      CALL FC   563 (
           ActReq                   := M    101.0,
           PLCNo                    := DB1575.DBW   14,
           SourceUnitNo             := 91,
           IsTUnit                  := FALSE,
           DstComDRec               := DB1575.CIP,
           RET_VAL                  := #wRetVal);


// ... CIP Distribution ------------- /

      L     DB1571.DBD   46;
      L     DB1945.DBD   10;
      ==D   ;
      JCN   CIP1;
      CALL FC   563 (
           ActReq                   := M    101.0,
           PLCNo                    := 3,
           SourceUnitNo             := 91,
           IsTUnit                  := FALSE,
           DstComDRec               := DB1575.CIP,
           RET_VAL                  := #wRetVal);

      CALL FC   563 (
           ActReq                   := M    101.0,
           PLCNo                    := 3,
           SourceUnitNo             := 94,
           IsTUnit                  := FALSE,
           DstComDRec               := DB1575.CIPDist,
           RET_VAL                  := #wRetVal);

      CALL SFC   20 (
           SRCBLK                   := DB1575.ToCIP,
           RET_VAL                  := #iRetVal,
           DSTBLK                   := DB502.ToCIP1);

CIP1: NOP   0;

      L     DB1571.DBD   46;
      L     DB1955.DBD   10;
      ==D   ;
      JCN   CIP2;
      CALL FC   563 (
           ActReq                   := M    101.0,
           PLCNo                    := 3,
           SourceUnitNo             := 92,
           IsTUnit                  := FALSE,
           DstComDRec               := DB1575.CIP,
           RET_VAL                  := #wRetVal);

      CALL FC   563 (
           ActReq                   := M    101.0,
           PLCNo                    := 3,
           SourceUnitNo             := 95,
           IsTUnit                  := FALSE,
           DstComDRec               := DB1575.CIPDist,
           RET_VAL                  := #wRetVal);

      CALL SFC   20 (
           SRCBLK                   := DB1575.ToCIP,
           RET_VAL                  := #iRetVal,
           DSTBLK                   := DB502.ToCIP2);
CIP2: NOP   0;

      L     DB1571.DBD   46;
      L     DB1965.DBD   10;
      ==D   ;
      JCN   CIP3;
      CALL FC   563 (
           ActReq                   := M    101.0,
           PLCNo                    := 3,
           SourceUnitNo             := 93,
           IsTUnit                  := FALSE,
           DstComDRec               := DB1575.CIP,
           RET_VAL                  := #wRetVal);

      CALL FC   563 (
           ActReq                   := M    101.0,
           PLCNo                    := 3,
           SourceUnitNo             := 96,
           IsTUnit                  := FALSE,
           DstComDRec               := DB1575.CIPDist,
           RET_VAL                  := #wRetVal);

      CALL SFC   20 (
           SRCBLK                   := DB1575.ToCIP,
           RET_VAL                  := #iRetVal,
           DSTBLK                   := DB502.ToCIP3);

CIP3: NOP   0;

//----------------------------------------
// Communication Water Tank
//----------------------------------------
// Current Tank ----------------------------
      CALL FC   950 (
           EquipmentNo              := DB1571.DBD  270,
           PLCNo                    := #iPLC,
           UnitNo                   := #iUnit);
      L     #iUnit;
      L     0;
      >I    ;
      JCN   T0xx;

      CALL FC   563 (
           ActReq                   := M    101.0,
           PLCNo                    := #iPLC,
           SourceUnitNo             := #iUnit,
           IsTUnit                  := FALSE,
           DstComDRec               := DB1575.SRC,
           RET_VAL                  := #wRetVal);
      JU    T0xy;
T0xx: NOP   0;
      T     #iTmp;
      CALL SFC   21 (
           BVAL                     := #iTmp,
           RET_VAL                  := #iRetVal,
           BLK                      := DB1575.SRC);
T0xy: NOP   0;

// Priority 1 -----------------------------
      CALL FC   950 (
           EquipmentNo              := DB1571.DBD  286,
           PLCNo                    := #iPLC,
           UnitNo                   := #iUnit);
      L     #iUnit;
      L     0;
      >I    ;
      JCN   T1xx;

      CALL FC   563 (
           ActReq                   := M    101.0,
           PLCNo                    := #iPLC,
           SourceUnitNo             := #iUnit,
           IsTUnit                  := FALSE,
           DstComDRec               := DB1575.SRC1,
           RET_VAL                  := #wRetVal);
      JU    T1xy;
T1xx: NOP   0;
      T     #iTmp;
      CALL SFC   21 (
           BVAL                     := #iTmp,
           RET_VAL                  := #iRetVal,
           BLK                      := DB1575.SRC1);
T1xy: NOP   0;

// Priority 2 ----------------------------
      CALL FC   950 (
           EquipmentNo              := DB1571.DBD  302,
           PLCNo                    := #iPLC,
           UnitNo                   := #iUnit);
      L     #iUnit;
      L     0;
      >I    ;
      JCN   T2xx;

      CALL FC   563 (
           ActReq                   := M    101.0,
           PLCNo                    := #iPLC,
           SourceUnitNo             := #iUnit,
           IsTUnit                  := FALSE,
           DstComDRec               := DB1575.SRC2,
           RET_VAL                  := #wRetVal);
      JU    T2xy;
T2xx: NOP   0;
      T     #iTmp;
      CALL SFC   21 (
           BVAL                     := #iTmp,
           RET_VAL                  := #iRetVal,
           BLK                      := DB1575.SRC2);
T2xy: NOP   0;

// Pririty 3 ----------------------------
      CALL FC   950 (
           EquipmentNo              := DB1571.DBD  318,
           PLCNo                    := #iPLC,
           UnitNo                   := #iUnit);
      L     #iUnit;
      L     0;
      >I    ;
      JCN   T3xx;

      CALL FC   563 (
           ActReq                   := M    101.0,
           PLCNo                    := #iPLC,
           SourceUnitNo             := #iUnit,
           IsTUnit                  := FALSE,
           DstComDRec               := DB1575.SRC3,
           RET_VAL                  := #wRetVal);
      JU    T3xy;
T3xx: NOP   0;
      T     #iTmp;
      CALL SFC   21 (
           BVAL                     := #iTmp,
           RET_VAL                  := #iRetVal,
           BLK                      := DB1575.SRC3);
T3xy: NOP   0;

//----------------------------------------
// Communication Brewhouse
//----------------------------------------
///   L     #U.Seq.Prop.Index0          // Destination
///   ITD
///   DTR
///   T     #rTmp

///  CALL  "Eq2PU"
//       EquipmentNo:=#rTmp
//       PLCNo      :=#iPLC
//       UnitNo     :=#iUnit

///  CALL  "UIT3"
//       ActReq      :="Clk1E"
//       PLCNo       :=#iPLC
//       SourceUnitNo:=#iUnit
//       IsTUnit     :=FALSE
//       DstComDRec  :="C04ComD".DST
//       RET_VAL     :=#wRetVal



NETWORK
TITLE =remote start

      SET   ;
// !!! insert correct condition of unit start !!!
      A     DB1571.DBX   15.0;
      A     DB1571.DBX   17.4;
      CLR   ;
      JCN   Strt;
      L     DB1575.DBD   10;
//L        L#-1;                            // Prid negative to start on its own
      T     #Prid;

      CALL FC    48 (
           UnitNo                   := #UnitNo,
           PrId                     := #Prid,
           Run                      := DB1571.DBX   17.4,
           PrIdTransfer             := TRUE,
           Start                    := TRUE,
           RetVal                   := #wRetVal);
Strt: NOP   0;
NETWORK
TITLE =external releases

      SET   ;
      =     DB2570.DBX  106.7;
      =     DB2570.DBX  426.7;
      =     DB2570.DBX  506.7;

NETWORK
TITLE =write own unit data

      SET   ;

//-- CIP Communication ---------------------------------------
      AN    DB1571.DBX   15.0;
//      AN "U057SeqD".Seq.PO.B30 // CIP Active (Slave)
      A     #ComCIP;
      JCN   NCIP;
//Conductivity CIP Return
      L     DB1575.DBD  150;
      T     DB1571.DBD  626;

//Temperature CIP Return
      L     DB1575.DBD  146;
      T     DB1571.DBD  594;

//CIP Prerun Pump SP

      CALL FC    45 (
           SFM                      := DB1571.DBD  686,
           Indexes                  := #SFM36);


      L     0.000000e+000;
      A     #SFM36.I01;
      =     DB1575.DBX  171.7;
      JCN   pfc;
      L     DB1571.DBD  654;
pfc:  NOP   0;
      A     #SFM36.I02;
      =     DB1575.DBX  172.0;
      JCN   ppc;
      L     DB1571.DBD  670;
ppc:  NOP   0;
      A     #SFM36.I03;
      =     DB1575.DBX  171.6;
      JCN   pxc;
      L     DB1571.DBD  574;
pxc:  NOP   0;
      T     DB1575.DBD  182;

//CIP Return
      L     DB1571.DBD  558;
      T     DB1575.DBD  186;
      L     DB1575.DBD  138;
      T     DB1571.DBD  562;

//CIP Prerun
      L     DB1571.DBD  542;
      T     DB1575.DBD  190;
      L     DB1575.DBD  142;
      T     DB1571.DBD  546;

// Write Own Data to CIP
      L     DB1575.DBD   10;
      T     DB1575.DBD  154;

      L     DB1575.DBW   14;
      T     DB1575.DBW  158;

      L     DB1575.DBW   16;
      T     DB1575.DBW  160;

      L     DB1575.DBW   18;
      T     DB1575.DBW  162;

      L     DB1575.DBW   20;
      T     DB1575.DBW  164;

      L     DB1575.DBW   22;
      T     DB1575.DBW  166;

      A     DB1575.DBX   24.0;
      =     DB1575.DBX  168.0;

      A     DB1575.DBX   24.1;
      =     DB1575.DBX  168.1;

      A     DB1575.DBX   24.2;
      =     DB1575.DBX  168.2;

      A     DB1575.DBX   24.3;
      =     DB1575.DBX  168.3;

      A     DB1575.DBX   24.4;
      =     DB1575.DBX  168.4;

      A     DB1575.DBX   24.5;
      =     DB1575.DBX  168.5;

      A     DB1575.DBX   24.6;
      =     DB1575.DBX  168.6;

      A     DB1575.DBX   24.7;
      =     DB1575.DBX  168.7;

// Copy Data to CIP
      CALL SFC   20 (
           SRCBLK                   := DB1575.ToCIP,
           RET_VAL                  := #iRetVal,
           DSTBLK                   := DB1575.ToCIP);

NCIP: NOP   0;

//Empty Signal
//A     "U057SpID".SpI.Sig //!!!! Insert correct Empty Signal !!!
      CLR   ;
      =     DB1575.DBX   26.5;

//Full Signal
//A     "U057SpID".SpI.Sig //!!!! Insert correct Full Signal !!!
      CLR   ;
      =     DB1575.DBX   26.2;

//CIP Program Selected
      A     #CIP;
      =     DB1575.DBX   27.1;

// Emergency Stop
      A     #EStopOK; //If needed add or replace with own SpI
      =     DB1575.DBX   27.0; //Emergency Stop OK

      L     DB1571.DBD  782; // Material
      T     DB1575.DBD   30;

      L     DB1571.DBD  270; // Current Water Tank Selection
      T     DB1575.DBD   34;

      L     DB1571.DBD  286; // Priority 1
      T     DB1575.DBD   38;

      L     DB1571.DBD  302; // Priority 2
      T     DB1575.DBD   42;

      L     DB1571.DBD  318; // Priority 3
      T     DB1575.DBD   46;

NETWORK
TITLE = read from other unit data



END_FUNCTION_BLOCK

FUNCTION_BLOCK FB 1579
TITLE =U057: Water Transfer Brewhouse
AUTHOR : Woermann
FAMILY : BOTEC_F1
NAME : Sim
VERSION : 0.1


VAR_TEMP
  CIP : BOOL ;	//CIP active
  xTmp : BOOL ;	//Temporary BOOL (free for general use)
  iTmp : INT ;	//Temporary INT (free for general use)
  rTmp : REAL ;	//Temporary REAL (free for general use)
  UnitNo : INT ;	//Unit Number
END_VAR
BEGIN
NETWORK
TITLE =General

      SET   ;
// get unit number ----------------------------------------------------------
      L     DB1570.DBW    0;
      T     #UnitNo;

// CIP ----------------------------------------------------------------------
      L     DB1571.DBD   54;
      L     0;
      <D    ;
      =     #CIP;

NETWORK
TITLE =Actuator

      A     DB1571.DBX   17.3;
      =     DB2570.DBX  105.3;
      =     DB2570.DBX  185.3;
      =     DB2570.DBX  265.3;
      =     DB2570.DBX  345.3;
      =     DB2570.DBX  505.3;


NETWORK
TITLE =Special Input

      A     DB1571.DBX   17.3;
      =     DB2571.DBX  141.3;
      =     DB2571.DBX  201.3;
      =     DB2571.DBX  261.3;
      =     DB2571.DBX  321.3;
      =     DB2571.DBX  381.3;

NETWORK
TITLE =Counter

      A     DB1571.DBX   17.3;
      A     M    101.0;


      CLR   ;
NETWORK
TITLE =Analog Input

      A     DB1571.DBX   17.3;

NETWORK
TITLE =Universal Value

      A     DB1571.DBX   17.3;
//      =     "U057UnVD".unv001.Sim;
//      =     "U057UnVD".unv002.Sim;
//      =     "U057UnVD".unv003.Sim;
//      =     "U057UnVD".unv004.Sim;

NETWORK
TITLE =PID

      A     DB1571.DBX   17.3;

NETWORK
TITLE =Message

      A     DB1571.DBX   17.3;
//      =     "U057MsgD".msg001.Sim;
//      =     "U057MsgD".msg002.Sim;
//      =     "U057MsgD".msg003.Sim;

NETWORK
TITLE =VLT

      A     DB1571.DBX   17.3;

END_FUNCTION_BLOCK

FUNCTION_BLOCK FB 1585
TITLE =U058: Water Transfer Syrup
FAMILY : BOTEC_F1
NAME : Comm
VERSION : 0.1


VAR_TEMP
  iRetVal : INT ;	//return value as integer
  wRetVal : WORD ;	//return value as word
  Run : BOOL ;	//Unit in "RUN" mode
  EStopOK : BOOL ;	//Emergency Stop OK
  CIP : BOOL ;	//CIP Program Selected
  ComCIP : BOOL ;	//Communication with CIP Active
  xTmp : BOOL ;	//Temporary BOOL (free for general use)
  iTmp : INT ;	//Temporary INT (free for general use)
  rTmp : REAL ;	//Temporary REAL (free for general use)
  dTmp : DINT ;	//Temporary DINT (free for general use)
  UnitNo : INT ;	//Unit Number
  EquipmentID : INT ;	//Equipment ID
  Prid : DINT ;	//Process ID
  SFM36 : STRUCT 	// CIP Pump Mode
   I00 : BOOL ;	// Off
   I01 : BOOL ;	// Flow
   I02 : BOOL ;	// Pressure
   I03 : BOOL ;	// Fix Speed
   I04 : BOOL ;
   I05 : BOOL ;
   I06 : BOOL ;
   I07 : BOOL ;
   I08 : BOOL ;
   I09 : BOOL ;
   I10 : BOOL ;
   I11 : BOOL ;
   I12 : BOOL ;
   I13 : BOOL ;
   I14 : BOOL ;
   I15 : BOOL ;
   I16 : BOOL ;
   I17 : BOOL ;
   I18 : BOOL ;
   I19 : BOOL ;
   I20 : BOOL ;
   I21 : BOOL ;
   I22 : BOOL ;
   I23 : BOOL ;
   I24 : BOOL ;
   I25 : BOOL ;
   I26 : BOOL ;
   I27 : BOOL ;
   I28 : BOOL ;
   I29 : BOOL ;
   I30 : BOOL ;
   I31 : BOOL ;
  END_STRUCT ;
  iPLC : INT ;
  iUnit : INT ;
END_VAR
BEGIN
NETWORK
TITLE =general

      SET   ;

// unit & equipment number ---------------------------------------------------
      L     DB1580.DBW    0;
      T     #UnitNo;

      L     DB1585.DBW   14;
      L     1000;
      *I    ;
      L     #UnitNo;
      +I    ;
      T     #EquipmentID;

// CIP ----------------------------------------------------------------------
      L     DB1585.DBW   18;
      L     0;
      <I    ;
      =     #CIP;

// Communicating Units-------------------------------------------------------
      L     DB1585.DBD   10;
      L     DB1585.DBD  106;
      ==D   ;
      =     #ComCIP;

// emergency OK -------------------------------------------------------------
      A     DB1585.DBX   75.0; //General Emergency Stop OK
      =     #EStopOK;

NETWORK
TITLE =read other unit's data

      SET   ;

// ... General Unit ----------/

      CALL FC   563 (
           ActReq                   := M    101.0,
           PLCNo                    := DB1585.DBW   14,
           SourceUnitNo             := 99,
           IsTUnit                  := FALSE,
           DstComDRec               := DB1585.GEN,
           RET_VAL                  := #wRetVal);


// ... CIP Unit ------------- /

      CALL FC   563 (
           ActReq                   := M    101.0,
           PLCNo                    := DB1585.DBW   14,
           SourceUnitNo             := 92,
           IsTUnit                  := FALSE,
           DstComDRec               := DB1585.CIP,
           RET_VAL                  := #wRetVal);


// ... CIP Distribution ------------- /
      L     DB1581.DBD   46;
      L     DB1955.DBD   10;
      ==D   ;
      JCN   CIP2;

      CALL FC   563 (
           ActReq                   := M    101.0,
           PLCNo                    := 3,
           SourceUnitNo             := 95,
           IsTUnit                  := FALSE,
           DstComDRec               := DB1585.CIPDist,
           RET_VAL                  := #wRetVal);

      CALL SFC   20 (
           SRCBLK                   := DB1585.ToCIP,
           RET_VAL                  := #iRetVal,
           DSTBLK                   := DB502.ToCIP2);
CIP2: NOP   0;

//----------------------------------------
// Communication Water Tank
//----------------------------------------
// Current Tank ----------------------------
      CALL FC   950 (
           EquipmentNo              := DB1581.DBD  270,
           PLCNo                    := #iPLC,
           UnitNo                   := #iUnit);
      L     #iUnit;
      L     0;
      >I    ;
      JCN   T0xx;
      CALL FC   563 (
           ActReq                   := M    101.0,
           PLCNo                    := #iPLC,
           SourceUnitNo             := #iUnit,
           IsTUnit                  := FALSE,
           DstComDRec               := DB1585.SRC,
           RET_VAL                  := #wRetVal);
      JU    T0xy;
T0xx: NOP   0;
      T     #iTmp;
      CALL SFC   21 (
           BVAL                     := #iTmp,
           RET_VAL                  := #iRetVal,
           BLK                      := DB1585.SRC);
T0xy: NOP   0;

// Priority 1 -----------------------------
      CALL FC   950 (
           EquipmentNo              := DB1581.DBD  286,
           PLCNo                    := #iPLC,
           UnitNo                   := #iUnit);
      L     #iUnit;
      L     0;
      >I    ;
      JCN   T1xx;

      CALL FC   563 (
           ActReq                   := M    101.0,
           PLCNo                    := #iPLC,
           SourceUnitNo             := #iUnit,
           IsTUnit                  := FALSE,
           DstComDRec               := DB1585.SRC1,
           RET_VAL                  := #wRetVal);
      JU    T1xy;
T1xx: NOP   0;
      T     #iTmp;
      CALL SFC   21 (
           BVAL                     := #iTmp,
           RET_VAL                  := #iRetVal,
           BLK                      := DB1585.SRC1);
T1xy: NOP   0;

// Priority 2 ----------------------------
      CALL FC   950 (
           EquipmentNo              := DB1581.DBD  302,
           PLCNo                    := #iPLC,
           UnitNo                   := #iUnit);
      L     #iUnit;
      L     0;
      >I    ;
      JCN   T2xx;

      CALL FC   563 (
           ActReq                   := M    101.0,
           PLCNo                    := #iPLC,
           SourceUnitNo             := #iUnit,
           IsTUnit                  := FALSE,
           DstComDRec               := DB1585.SRC2,
           RET_VAL                  := #wRetVal);
      JU    T2xy;
T2xx: NOP   0;
      T     #iTmp;
      CALL SFC   21 (
           BVAL                     := #iTmp,
           RET_VAL                  := #iRetVal,
           BLK                      := DB1585.SRC2);
T2xy: NOP   0;

// Pririty 3 ----------------------------
      CALL FC   950 (
           EquipmentNo              := DB1581.DBD  318,
           PLCNo                    := #iPLC,
           UnitNo                   := #iUnit);
      L     #iUnit;
      L     0;
      >I    ;
      JCN   T3xx;

      CALL FC   563 (
           ActReq                   := M    101.0,
           PLCNo                    := #iPLC,
           SourceUnitNo             := #iUnit,
           IsTUnit                  := FALSE,
           DstComDRec               := DB1585.SRC3,
           RET_VAL                  := #wRetVal);
      JU    T3xy;
T3xx: NOP   0;
      T     #iTmp;
      CALL SFC   21 (
           BVAL                     := #iTmp,
           RET_VAL                  := #iRetVal,
           BLK                      := DB1585.SRC3);
T3xy: NOP   0;


// Sirupraum
      CALL FC   563 (
           ActReq                   := M    101.0,
           PLCNo                    := 1,
           SourceUnitNo             := 8,
           IsTUnit                  := FALSE,
           DstComDRec               := DB1585.DST,
           RET_VAL                  := #wRetVal);

NETWORK
TITLE =remote start

      SET   ;
// !!! insert correct condition of unit start !!!
      A     DB1581.DBX   15.0;
      A     DB1581.DBX   17.4;
      CLR   ;
      JCN   Strt;
      L     DB1585.DBD   10;
//L        L#-1;                            // Prid negative to start on its own
      T     #Prid;

      CALL FC    48 (
           UnitNo                   := #UnitNo,
           PrId                     := #Prid,
           Run                      := DB1581.DBX   17.4,
           PrIdTransfer             := TRUE,
           Start                    := TRUE,
           RetVal                   := #wRetVal);
Strt: NOP   0;
NETWORK
TITLE =external releases

      SET   ;
      =     DB2580.DBX  106.7;
      =     DB2580.DBX  186.7;
      =     DB2580.DBX  266.7;
NETWORK
TITLE =write own unit data

      SET   ;

//-- CIP Communication ---------------------------------------
      AN    DB1581.DBX   15.0;
//      AN "U058SeqD".Seq.PO.B30 // CIP Active (Slave)
      A     #ComCIP;
      JCN   NCIP;
//Conductivity CIP Return
      L     DB1585.DBD  150;
      T     DB1581.DBD  626;

//Temperature CIP Return
      L     DB1585.DBD  146;
      T     DB1581.DBD  594;

//CIP Prerun Pump SP

      CALL FC    45 (
           SFM                      := DB1581.DBD  686,
           Indexes                  := #SFM36);


      L     0.000000e+000;
      A     #SFM36.I01;
      =     DB1585.DBX  171.7;
      JCN   pfc;
      L     DB1581.DBD  654;
pfc:  NOP   0;
      A     #SFM36.I02;
      =     DB1585.DBX  172.0;
      JCN   ppc;
      L     DB1581.DBD  670;
ppc:  NOP   0;
      A     #SFM36.I03;
      =     DB1585.DBX  171.6;
      JCN   pxc;
      L     DB1581.DBD  574;
pxc:  NOP   0;
      T     DB1585.DBD  182;

//CIP Return
      L     DB1581.DBD  558;
      T     DB1585.DBD  186;
      L     DB1585.DBD  138;
      T     DB1581.DBD  562;

//CIP Prerun
      L     DB1581.DBD  542;
      T     DB1585.DBD  190;
      L     DB1585.DBD  142;
      T     DB1581.DBD  546;

// Write Own Data to CIP
      L     DB1585.DBD   10;
      T     DB1585.DBD  154;

      L     DB1585.DBW   14;
      T     DB1585.DBW  158;

      L     DB1585.DBW   16;
      T     DB1585.DBW  160;

      L     DB1585.DBW   18;
      T     DB1585.DBW  162;

      L     DB1585.DBW   20;
      T     DB1585.DBW  164;

      L     DB1585.DBW   22;
      T     DB1585.DBW  166;

      A     DB1585.DBX   24.0;
      =     DB1585.DBX  168.0;

      A     DB1585.DBX   24.1;
      =     DB1585.DBX  168.1;

      A     DB1585.DBX   24.2;
      =     DB1585.DBX  168.2;

      A     DB1585.DBX   24.3;
      =     DB1585.DBX  168.3;

      A     DB1585.DBX   24.4;
      =     DB1585.DBX  168.4;

      A     DB1585.DBX   24.5;
      =     DB1585.DBX  168.5;

      A     DB1585.DBX   24.6;
      =     DB1585.DBX  168.6;

      A     DB1585.DBX   24.7;
      =     DB1585.DBX  168.7;

// Copy Data to CIP
      CALL SFC   20 (
           SRCBLK                   := DB1585.ToCIP,
           RET_VAL                  := #iRetVal,
           DSTBLK                   := DB502.ToCIP2);

NCIP: NOP   0;

//Empty Signal
//A     "U058SpID".SpI.Sig //!!!! Insert correct Empty Signal !!!
      CLR   ;
      =     DB1585.DBX   26.5;

//Full Signal
//A     "U058SpID".SpI.Sig //!!!! Insert correct Full Signal !!!
      CLR   ;
      =     DB1585.DBX   26.2;

//CIP Program Selected
      A     #CIP;
      =     DB1585.DBX   27.1;

// Emergency Stop
      A     #EStopOK; //If needed add or replace with own SpI
      =     DB1585.DBX   27.0; //Emergency Stop OK

// Weitere Signale
      L     DB1581.DBD  782; // Material
      T     DB1585.DBD   30;

      L     DB1581.DBD  270; // Current Water Tank Selection
      T     DB1585.DBD   34;

      L     DB1581.DBD  286; // Priority 1
      T     DB1585.DBD   38;

      L     DB1581.DBD  302; // Priority 2
      T     DB1585.DBD   42;

      L     DB1581.DBD  318; // Priority 3
      T     DB1585.DBD   46;



      A     DB1585.DBX  458.1;
      ON    DB5030.DBX  182.5;
      ON    DB5050.DBX  182.5;
      ON    DB5070.DBX  182.5;
      ON    DB5090.DBX  182.5;
      ON    DB5120.DBX  182.5;
      ON    DB5140.DBX  182.5;
      =     DB1585.DBX   26.3;


NETWORK
TITLE = read from other unit data



END_FUNCTION_BLOCK

FUNCTION_BLOCK FB 1589
TITLE =U058: Water Transfer Syrup
AUTHOR : Woermann
FAMILY : BOTEC_F1
NAME : Sim
VERSION : 0.1


VAR_TEMP
  CIP : BOOL ;	//CIP active
  xTmp : BOOL ;	//Temporary BOOL (free for general use)
  iTmp : INT ;	//Temporary INT (free for general use)
  rTmp : REAL ;	//Temporary REAL (free for general use)
  UnitNo : INT ;	//Unit Number
END_VAR
BEGIN
NETWORK
TITLE =General

      SET   ;
// get unit number ----------------------------------------------------------
      L     DB1580.DBW    0;
      T     #UnitNo;

// CIP ----------------------------------------------------------------------
      L     DB1581.DBD   54;
      L     0;
      <D    ;
      =     #CIP;

NETWORK
TITLE =Actuator

      A     DB1581.DBX   17.3;
      =     DB2580.DBX  105.3;
      =     DB2580.DBX  185.3;
      =     DB2580.DBX  265.3;
      =     DB2580.DBX  505.3;

NETWORK
TITLE =Special Input

      A     DB1581.DBX   17.3;
      =     DB2581.DBX  141.3;
      =     DB2581.DBX  201.3;


NETWORK
TITLE =Counter

      A     DB1581.DBX   17.3;
      A     M    101.0;


      CLR   ;
NETWORK
TITLE =Analog Input

      A     DB1581.DBX   17.3;
      =     DB2583.DBX  141.3;

NETWORK
TITLE =Universal Value

      A     DB1581.DBX   17.3;
//      =     "U058UnVD".unv001.Sim;
//      =     "U058UnVD".unv002.Sim;
//      =     "U058UnVD".unv003.Sim;
//      =     "U058UnVD".unv004.Sim;

NETWORK
TITLE =PID

      A     DB1581.DBX   17.3;
//      =     "U058PIDD".SR_P1_PID.Ign;

NETWORK
TITLE =Message

      A     DB1581.DBX   17.3;
//      =     "U058MsgD".msg001.Sim;
//      =     "U058MsgD".msg002.Sim;
//      =     "U058MsgD".msg003.Sim;

NETWORK
TITLE =VLT

      A     DB1581.DBX   17.3;

END_FUNCTION_BLOCK

FUNCTION_BLOCK FB 1595
TITLE =U059: Molchwasser
FAMILY : BOTEC_F1
NAME : U059Comm
VERSION : 0.1


VAR_TEMP
  iRetVal : INT ;	//return value as integer
  wRetVal : WORD ;	//return value as word
  Run : BOOL ;	//Unit in "RUN" mode
  EStopOK : BOOL ;	//Emergency Stop OK
  CIP : BOOL ;	//CIP Program Selected
  ComCIP : BOOL ;	//Communication with CIP Active
  xTmp : BOOL ;	//Temporary BOOL (free for general use)
  iTmp : INT ;	//Temporary INT (free for general use)
  rTmp : REAL ;	//Temporary REAL (free for general use)
  dTmp : DINT ;	//Temporary DINT (free for general use)
  UnitNo : INT ;	//Unit Number
  EquipmentID : INT ;	//Equipment ID
  Prid : DINT ;	//Process ID
  SFM36 : STRUCT 	// CIP Pump Mode
   I00 : BOOL ;	// Off
   I01 : BOOL ;	// Flow
   I02 : BOOL ;	// Pressure
   I03 : BOOL ;	// Fix Speed
   I04 : BOOL ;
   I05 : BOOL ;
   I06 : BOOL ;
   I07 : BOOL ;
   I08 : BOOL ;
   I09 : BOOL ;
   I10 : BOOL ;
   I11 : BOOL ;
   I12 : BOOL ;
   I13 : BOOL ;
   I14 : BOOL ;
   I15 : BOOL ;
   I16 : BOOL ;
   I17 : BOOL ;
   I18 : BOOL ;
   I19 : BOOL ;
   I20 : BOOL ;
   I21 : BOOL ;
   I22 : BOOL ;
   I23 : BOOL ;
   I24 : BOOL ;
   I25 : BOOL ;
   I26 : BOOL ;
   I27 : BOOL ;
   I28 : BOOL ;
   I29 : BOOL ;
   I30 : BOOL ;
   I31 : BOOL ;
  END_STRUCT ;
END_VAR
BEGIN
NETWORK
TITLE =general

      SET   ;

// unit & equipment number ---------------------------------------------------
      L     DB1590.DBW    0;
      T     #UnitNo;

      L     DB1595.DBW   14;
      L     1000;
      *I    ;
      L     #UnitNo;
      +I    ;
      T     #EquipmentID;

// CIP ----------------------------------------------------------------------
      L     DB1595.DBW   18;
      L     0;
      <I    ;
      =     #CIP;

// Communicating Units-------------------------------------------------------
      L     DB1595.DBD   10;
      L     DB1595.DBD  106;
      ==D   ;
      =     #ComCIP;

// emergency OK -------------------------------------------------------------
      A     DB1595.DBX   75.0; //General Emergency Stop OK
      =     #EStopOK;

NETWORK
TITLE =read other unit's data

      SET   ;

// ... General Unit ----------/

      CALL FC   563 (
           ActReq                   := M    101.0,
           PLCNo                    := 3,
           SourceUnitNo             := 99,
           IsTUnit                  := FALSE,
           DstComDRec               := DB1595.GEN,
           RET_VAL                  := #wRetVal);


NETWORK
TITLE =remote start
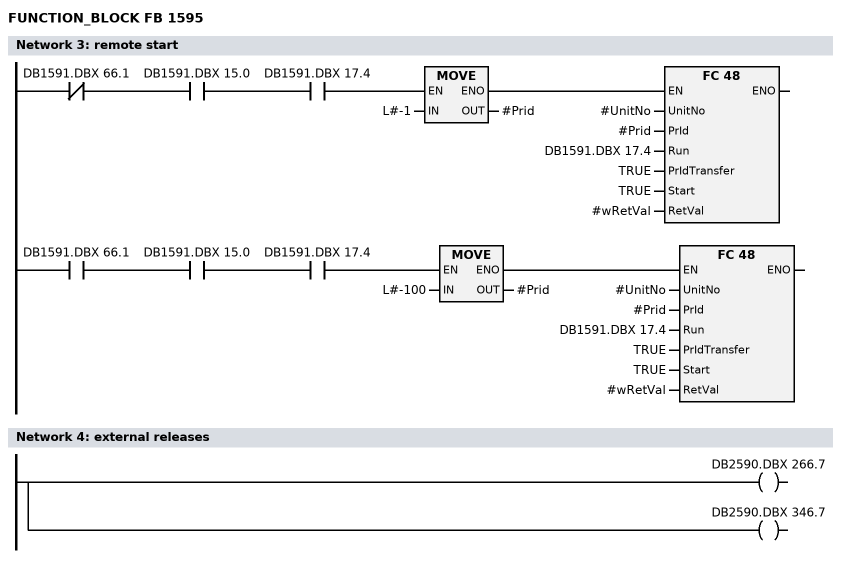

      SET   ;
      AN    DB1591.DBX   66.1;
      A     DB1591.DBX   15.0;
      A     DB1591.DBX   17.4;
      JCN   Strt;
      L     L#-1; // Prid negative to start on its own
      T     #Prid;

      CALL FC    48 (
           UnitNo                   := #UnitNo,
           PrId                     := #Prid,
           Run                      := DB1591.DBX   17.4,
           PrIdTransfer             := TRUE,
           Start                    := TRUE,
           RetVal                   := #wRetVal);
Strt: NOP   0;

      A     DB1591.DBX   66.1;
      A     DB1591.DBX   15.0;
      A     DB1591.DBX   17.4;
      JCN   Str2;
      L     L#-100; // Prid negative to start on its own
      T     #Prid;

      CALL FC    48 (
           UnitNo                   := #UnitNo,
           PrId                     := #Prid,
           Run                      := DB1591.DBX   17.4,
           PrIdTransfer             := TRUE,
           Start                    := TRUE,
           RetVal                   := #wRetVal);
Str2: NOP   0;

NETWORK
TITLE =external releases

      SET   ;
      =     DB2590.DBX  266.7;
      =     DB2590.DBX  346.7;
NETWORK
TITLE =write own unit data

      SET   ;

//-- CIP Communication ---------------------------------------
      AN    DB1591.DBX   15.0;
//      AN "U059SeqD".Seq.PO.B30 // CIP Active (Slave)
      A     #ComCIP;
      JCN   NCIP;
//Conductivity CIP Return
      L     DB1595.DBD  150;
      T     DB1591.DBD  626;

//Temperature CIP Return
      L     DB1595.DBD  146;
      T     DB1591.DBD  594;

//CIP Prerun Pump SP

      CALL FC    45 (
           SFM                      := DB1591.DBD  686,
           Indexes                  := #SFM36);


      L     0.000000e+000;
      A     #SFM36.I01;
      =     DB1595.DBX  171.7;
      JCN   pfc;
      L     DB1591.DBD  654;
pfc:  NOP   0;
      A     #SFM36.I02;
      =     DB1595.DBX  172.0;
      JCN   ppc;
      L     DB1591.DBD  670;
ppc:  NOP   0;
      A     #SFM36.I03;
      =     DB1595.DBX  171.6;
      JCN   pxc;
      L     DB1591.DBD  574;
pxc:  NOP   0;
      T     DB1595.DBD  182;

//CIP Return
      L     DB1591.DBD  558;
      T     DB1595.DBD  186;
      L     DB1595.DBD  138;
      T     DB1591.DBD  562;

//CIP Prerun
      L     DB1591.DBD  542;
      T     DB1595.DBD  190;
      L     DB1595.DBD  142;
      T     DB1591.DBD  546;

// Write Own Data to CIP
      L     DB1595.DBD   10;
      T     DB1595.DBD  154;

      L     DB1595.DBW   14;
      T     DB1595.DBW  158;

      L     DB1595.DBW   16;
      T     DB1595.DBW  160;

      L     DB1595.DBW   18;
      T     DB1595.DBW  162;

      L     DB1595.DBW   20;
      T     DB1595.DBW  164;

      L     DB1595.DBW   22;
      T     DB1595.DBW  166;

      A     DB1595.DBX   24.0;
      =     DB1595.DBX  168.0;

      A     DB1595.DBX   24.1;
      =     DB1595.DBX  168.1;

      A     DB1595.DBX   24.2;
      =     DB1595.DBX  168.2;

      A     DB1595.DBX   24.3;
      =     DB1595.DBX  168.3;

      A     DB1595.DBX   24.4;
      =     DB1595.DBX  168.4;

      A     DB1595.DBX   24.5;
      =     DB1595.DBX  168.5;

      A     DB1595.DBX   24.6;
      =     DB1595.DBX  168.6;

      A     DB1595.DBX   24.7;
      =     DB1595.DBX  168.7;

// Copy Data to CIP
      CALL SFC   20 (
           SRCBLK                   := DB1595.ToCIP,
           RET_VAL                  := #iRetVal,
           DSTBLK                   := DB1595.ToCIP);

NCIP: NOP   0;

//Empty Signal
//A     "U059SpID".SpI.Sig //!!!! Insert correct Empty Signal !!!
      CLR   ;
      =     DB1595.DBX   26.5;

//Full Signal
//A     "U059SpID".SpI.Sig //!!!! Insert correct Full Signal !!!
      CLR   ;
      =     DB1595.DBX   26.2;

//CIP Program Selected
      A     #CIP;
      =     DB1595.DBX   27.1;

// Emergency Stop
      A     #EStopOK; //If needed add or replace with own SpI
      =     DB1595.DBX   27.0; //Emergency Stop OK


NETWORK
TITLE = read from other unit data



END_FUNCTION_BLOCK

FUNCTION_BLOCK FB 1599
TITLE =U059: Pig Water
AUTHOR : Woermann
FAMILY : BOTEC_F1
NAME : Sim
VERSION : 0.1


VAR_TEMP
  CIP : BOOL ;	//CIP active
  xTmp : BOOL ;	//Temporary BOOL (free for general use)
  iTmp : INT ;	//Temporary INT (free for general use)
  rTmp : REAL ;	//Temporary REAL (free for general use)
  UnitNo : INT ;	//Unit Number
END_VAR
BEGIN
NETWORK
TITLE =General

      SET   ;
// get unit number ----------------------------------------------------------
      L     DB1590.DBW    0;
      T     #UnitNo;

// CIP ----------------------------------------------------------------------
      L     DB1591.DBD   54;
      L     0;
      <D    ;
      =     #CIP;

NETWORK
TITLE =Actuator

      A     DB1591.DBX   17.3;
      =     DB2590.DBX  105.3;
      =     DB2590.DBX  185.3;

NETWORK
TITLE =Special Input

      A     DB1591.DBX   17.3;



NETWORK
TITLE =Counter

      A     DB1591.DBX   17.3;
      A     M    101.0;


      CLR   ;
NETWORK
TITLE =Analog Input

      A     DB1591.DBX   17.3;


NETWORK
TITLE =Universal Value

      A     DB1591.DBX   17.3;
//      =     "U059UnVD".unv001.Sim;
//      =     "U059UnVD".unv002.Sim;
//      =     "U059UnVD".unv003.Sim;
//      =     "U059UnVD".unv004.Sim;

NETWORK
TITLE =PID

      A     DB1591.DBX   17.3;

NETWORK
TITLE =Message

      A     DB1591.DBX   17.3;
//    =     "U059MsgD".msg001.Sim
//     =     "U059MsgD".msg002.Sim
//      =     "U059MsgD".msg003.Sim

NETWORK
TITLE =VLT

      A     DB1591.DBX   17.3;

END_FUNCTION_BLOCK

FUNCTION_BLOCK FB 1635
TITLE =U063: Packaging Plant 3
FAMILY : BOTEC_F1
NAME : Comm
VERSION : 0.1


VAR_TEMP
  iRetVal : INT ;	//return value as integer
  wRetVal : WORD ;	//return value as word
  Run : BOOL ;	//Unit in "RUN" mode
  EStopOK : BOOL ;	//Emergency Stop OK
  CIP : BOOL ;	//CIP Program Selected
  ComCIP : BOOL ;	//Communication with CIP Active
  xTmp : BOOL ;	//Temporary BOOL (free for general use)
  iTmp : INT ;	//Temporary INT (free for general use)
  rTmp : REAL ;	//Temporary REAL (free for general use)
  dTmp : DINT ;	//Temporary DINT (free for general use)
  UnitNo : INT ;	//Unit Number
  EquipmentID : INT ;	//Equipment ID
  Prid : DINT ;	//Process ID
  SFM36 : STRUCT 	// CIP Pump Mode
   I00 : BOOL ;	// Off
   I01 : BOOL ;	// Flow
   I02 : BOOL ;	// Pressure
   I03 : BOOL ;	// Fix Speed
   I04 : BOOL ;
   I05 : BOOL ;
   I06 : BOOL ;
   I07 : BOOL ;
   I08 : BOOL ;
   I09 : BOOL ;
   I10 : BOOL ;
   I11 : BOOL ;
   I12 : BOOL ;
   I13 : BOOL ;
   I14 : BOOL ;
   I15 : BOOL ;
   I16 : BOOL ;
   I17 : BOOL ;
   I18 : BOOL ;
   I19 : BOOL ;
   I20 : BOOL ;
   I21 : BOOL ;
   I22 : BOOL ;
   I23 : BOOL ;
   I24 : BOOL ;
   I25 : BOOL ;
   I26 : BOOL ;
   I27 : BOOL ;
   I28 : BOOL ;
   I29 : BOOL ;
   I30 : BOOL ;
   I31 : BOOL ;
  END_STRUCT ;
END_VAR
BEGIN
NETWORK
TITLE =general

      SET   ;

// unit & equipment number ---------------------------------------------------
      L     DB1630.DBW    0;
      T     #UnitNo;

      L     DB1635.DBW   14;
      L     1000;
      *I    ;
      L     #UnitNo;
      +I    ;
      T     #EquipmentID;

// CIP ----------------------------------------------------------------------
      L     DB1635.DBW   18;
      L     0;
      <I    ;
      =     #CIP;

// Communicating Units-------------------------------------------------------
      L     DB1635.DBD   10;
      L     DB1635.DBD  106;
      ==D   ;
      =     #ComCIP;

// emergency OK -------------------------------------------------------------
      A     DB1635.DBX   75.0; //General Emergency Stop OK
      =     #EStopOK;

NETWORK
TITLE =read other unit's data

      SET   ;

// ... General Unit ----------/

      CALL FC   563 (
           ActReq                   := M    101.0,
           PLCNo                    := DB1635.DBW   14,
           SourceUnitNo             := 99,
           IsTUnit                  := FALSE,
           DstComDRec               := DB1635.GEN,
           RET_VAL                  := #wRetVal);


// ... CIP Unit ------------- /
      L     DB1631.DBD   46; // Select
      L     L#0; // Off
      ==D   ;
      JC    ELS1;
      TAK   ;
      L     DB1925.DBD   10; // CIP 2
      ==D   ;
      JC    M102;
      JU    ELS1;
M102: NOP   0; // Do 2
      CALL FC   563 (
           ActReq                   := M    101.0,
           PLCNo                    := 3,
           SourceUnitNo             := 92,
           IsTUnit                  := FALSE,
           DstComDRec               := DB1635.CIP,
           RET_VAL                  := #wRetVal);

      JU    FIN1;
ELS1: L     0;
      T     #iTmp;
      CALL SFC   21 (
           BVAL                     := #iTmp,
           RET_VAL                  := #iRetVal,
           BLK                      := DB1635.CIP);

FIN1: NOP   0;

NETWORK
TITLE =remote start
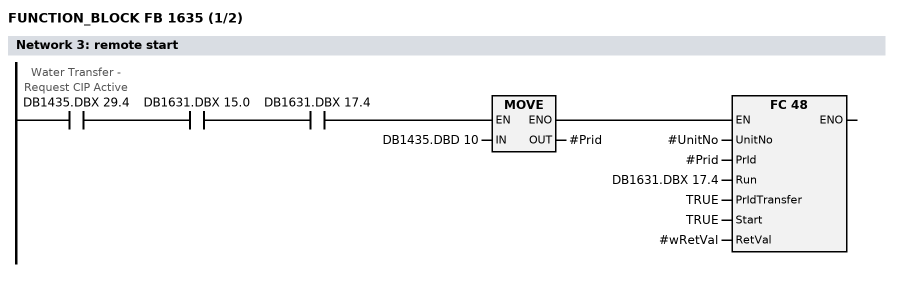

      SET   ;
      A     DB1435.DBX   29.4; // Water Transfer - Request CIP Active
      A     DB1631.DBX   15.0;
      A     DB1631.DBX   17.4;

      JCN   Strt;
      L     DB1435.DBD   10;
      T     #Prid;


      CALL FC    48 (
           UnitNo                   := #UnitNo,
           PrId                     := #Prid,
           Run                      := DB1631.DBX   17.4,
           PrIdTransfer             := TRUE,
           Start                    := TRUE,
           RetVal                   := #wRetVal);
Strt: NOP   0;
NETWORK
TITLE =external releases
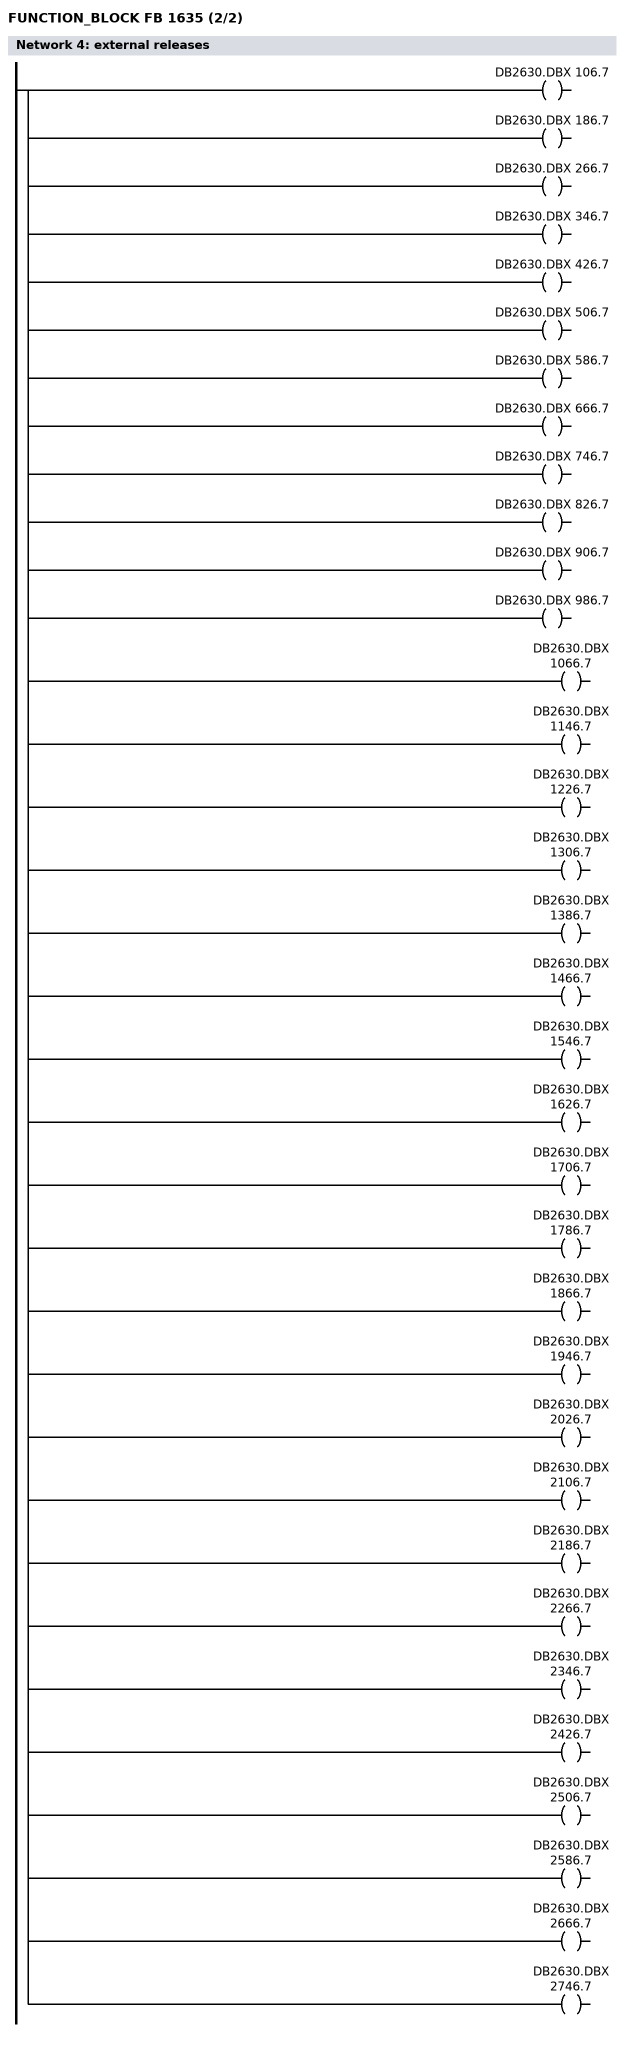

      SET   ;
      =     DB2630.DBX  106.7;
      =     DB2630.DBX  186.7;
      =     DB2630.DBX  266.7;
      =     DB2630.DBX  346.7;
      =     DB2630.DBX  426.7;
      =     DB2630.DBX  506.7;
      =     DB2630.DBX  586.7;
      =     DB2630.DBX  666.7;
      =     DB2630.DBX  746.7;
      =     DB2630.DBX  826.7;
      =     DB2630.DBX  906.7;
      =     DB2630.DBX  986.7;
      =     DB2630.DBX 1066.7;
      =     DB2630.DBX 1146.7;
      =     DB2630.DBX 1226.7;
      =     DB2630.DBX 1306.7;
      =     DB2630.DBX 1386.7;
      =     DB2630.DBX 1466.7;
      =     DB2630.DBX 1546.7;
      =     DB2630.DBX 1626.7;
      =     DB2630.DBX 1706.7;
      =     DB2630.DBX 1786.7;
      =     DB2630.DBX 1866.7;
      =     DB2630.DBX 1946.7;
      =     DB2630.DBX 2026.7;
      =     DB2630.DBX 2106.7;
      =     DB2630.DBX 2186.7;
      =     DB2630.DBX 2266.7;
      =     DB2630.DBX 2346.7;
      =     DB2630.DBX 2426.7;
      =     DB2630.DBX 2506.7;
      =     DB2630.DBX 2586.7;
      =     DB2630.DBX 2666.7;
      =     DB2630.DBX 2746.7;

NETWORK
TITLE =write own unit data

      SET   ;

//-- CIP Communication ---------------------------------------
      AN    DB1631.DBX   15.0;
      AN    DB1631.DBX 1233.6; // CIP Active (Slave)
      A     #ComCIP;
      JCN   NCIP;
//Conductivity CIP Return
      L     DB1635.DBD  150;
      T     DB1631.DBD  626;

//Temperature CIP Return
      L     DB1635.DBD  146;
      T     DB1631.DBD  594;

//CIP Prerun Pump SP

      CALL FC    45 (
           SFM                      := DB1631.DBD  686,
           Indexes                  := #SFM36);


      L     0.000000e+000;
      A     #SFM36.I01;
      =     DB1635.DBX  171.7;
      JCN   pfc;
      L     DB1631.DBD  654;
pfc:  NOP   0;
      A     #SFM36.I02;
      =     DB1635.DBX  172.0;
      JCN   ppc;
      L     DB1631.DBD  670;
ppc:  NOP   0;
      A     #SFM36.I03;
      =     DB1635.DBX  171.6;
      JCN   pxc;
      L     DB1631.DBD  574;
pxc:  NOP   0;
      T     DB1635.DBD  182;

//CIP Return
      L     DB1631.DBD  558;
      T     DB1635.DBD  186;
      L     DB1635.DBD  138;
      T     DB1631.DBD  562;

//CIP Prerun
      L     DB1631.DBD  542;
      T     DB1635.DBD  190;
      L     DB1635.DBD  142;
      T     DB1631.DBD  546;

// Write Own Data to CIP
      L     DB1635.DBD   10;
      T     DB1635.DBD  154;

      L     DB1635.DBW   14;
      T     DB1635.DBW  158;

      L     DB1635.DBW   16;
      T     DB1635.DBW  160;

      L     DB1635.DBW   18;
      T     DB1635.DBW  162;

      L     DB1635.DBW   20;
      T     DB1635.DBW  164;

      L     DB1635.DBW   22;
      T     DB1635.DBW  166;

      A     DB1635.DBX   24.0;
      =     DB1635.DBX  168.0;

      A     DB1635.DBX   24.1;
      =     DB1635.DBX  168.1;

      A     DB1635.DBX   24.2;
      =     DB1635.DBX  168.2;

      A     DB1635.DBX   24.3;
      =     DB1635.DBX  168.3;

      A     DB1635.DBX   24.4;
      =     DB1635.DBX  168.4;

      A     DB1635.DBX   24.5;
      =     DB1635.DBX  168.5;

      A     DB1635.DBX   24.6;
      =     DB1635.DBX  168.6;

      A     DB1635.DBX   24.7;
      =     DB1635.DBX  168.7;

// Copy Data to CIP
      CALL SFC   20 (
           SRCBLK                   := DB1635.ToCIP,
           RET_VAL                  := #iRetVal,
           DSTBLK                   := DB1635.ToCIP);

NCIP: NOP   0;

//Empty Signal
//A     "U063SpID".SpI.Sig //!!!! Insert correct Empty Signal !!!
      CLR   ;
      =     DB1635.DBX   26.5;

//Full Signal
//A     "U063SpID".SpI.Sig //!!!! Insert correct Full Signal !!!
      CLR   ;
      =     DB1635.DBX   26.2;

//CIP Program Selected
      A     #CIP;
      =     DB1635.DBX   27.1;

// Emergency Stop
      A     #EStopOK; //If needed add or replace with own SpI
      =     DB1635.DBX   27.0; //Emergency Stop OK


NETWORK
TITLE = read from other unit data

      A     M    100.7;
      =     Q    946.0;
      =     Q    986.0;

      SET   ;
      =     DB2630.DBX  748.2;

END_FUNCTION_BLOCK

FUNCTION_BLOCK FB 1639
TITLE =U063: Packaging Plant 3
AUTHOR : Woermann
FAMILY : BOTEC_F1
NAME : Sim
VERSION : 0.1


VAR_TEMP
  CIP : BOOL ;	//CIP active
  xTmp : BOOL ;	//Temporary BOOL (free for general use)
  iTmp : INT ;	//Temporary INT (free for general use)
  rTmp : REAL ;	//Temporary REAL (free for general use)
  UnitNo : INT ;	//Unit Number
END_VAR
BEGIN
NETWORK
TITLE =General

      SET   ;
// get unit number ----------------------------------------------------------
      L     DB1630.DBW    0;
      T     #UnitNo;

// CIP ----------------------------------------------------------------------
      L     DB1631.DBD   54;
      L     0;
      <D    ;
      =     #CIP;

NETWORK
TITLE =Actuator

      A     DB1631.DBX   17.3;
      =     DB2630.DBX  105.3;
      =     DB2630.DBX  185.3;

NETWORK
TITLE =Special Input

      A     DB1631.DBX   17.3;
      =     DB2631.DBX  141.3;
      =     DB2631.DBX  201.3;
NETWORK
TITLE =Counter

      A     DB1631.DBX   17.3;
      A     M    101.0;


      CLR   ;
NETWORK
TITLE =Analog Input

      A     DB1631.DBX   17.3;

NETWORK
TITLE =Universal Value

      A     DB1631.DBX   17.3;
//      =     "U063UnVD".unv001.Sim;
//      =     "U063UnVD".unv002.Sim;
//      =     "U063UnVD".unv003.Sim;
//      =     "U063UnVD".unv004.Sim;

NETWORK
TITLE =PID

      A     DB1631.DBX   17.3;

NETWORK
TITLE =Message

      A     DB1631.DBX   17.3;
//      =     "U063MsgD".msg001.Sim;
//      =     "U063MsgD".msg002.Sim;
//      =     "U063MsgD".msg003.Sim;

NETWORK
TITLE =VLT

      A     DB1631.DBX   17.3;

END_FUNCTION_BLOCK

FUNCTION_BLOCK FB 1655
TITLE =U065: Packaging Plant 5
FAMILY : BOTEC_F1
NAME : Comm
VERSION : 0.1


VAR_TEMP
  iRetVal : INT ;	//return value as integer
  wRetVal : WORD ;	//return value as word
  Run : BOOL ;	//Unit in "RUN" mode
  EStopOK : BOOL ;	//Emergency Stop OK
  CIP : BOOL ;	//CIP Program Selected
  ComCIP : BOOL ;	//Communication with CIP Active
  xTmp : BOOL ;	//Temporary BOOL (free for general use)
  iTmp : INT ;	//Temporary INT (free for general use)
  rTmp : REAL ;	//Temporary REAL (free for general use)
  dTmp : DINT ;	//Temporary DINT (free for general use)
  UnitNo : INT ;	//Unit Number
  EquipmentID : INT ;	//Equipment ID
  Prid : DINT ;	//Process ID
  SFM36 : STRUCT 	// CIP Pump Mode
   I00 : BOOL ;	// Off
   I01 : BOOL ;	// Flow
   I02 : BOOL ;	// Pressure
   I03 : BOOL ;	// Fix Speed
   I04 : BOOL ;
   I05 : BOOL ;
   I06 : BOOL ;
   I07 : BOOL ;
   I08 : BOOL ;
   I09 : BOOL ;
   I10 : BOOL ;
   I11 : BOOL ;
   I12 : BOOL ;
   I13 : BOOL ;
   I14 : BOOL ;
   I15 : BOOL ;
   I16 : BOOL ;
   I17 : BOOL ;
   I18 : BOOL ;
   I19 : BOOL ;
   I20 : BOOL ;
   I21 : BOOL ;
   I22 : BOOL ;
   I23 : BOOL ;
   I24 : BOOL ;
   I25 : BOOL ;
   I26 : BOOL ;
   I27 : BOOL ;
   I28 : BOOL ;
   I29 : BOOL ;
   I30 : BOOL ;
   I31 : BOOL ;
  END_STRUCT ;
END_VAR
BEGIN
NETWORK
TITLE =general

      SET   ;

// unit & equipment number ---------------------------------------------------
      L     DB1650.DBW    0;
      T     #UnitNo;

      L     DB1655.DBW   14;
      L     1000;
      *I    ;
      L     #UnitNo;
      +I    ;
      T     #EquipmentID;

// CIP ----------------------------------------------------------------------
      L     DB1655.DBW   18;
      L     0;
      <I    ;
      =     #CIP;

// Communicating Units-------------------------------------------------------
      L     DB1655.DBD   10;
      L     DB1655.DBD  106;
      ==D   ;
      =     #ComCIP;

// emergency OK -------------------------------------------------------------
      A     DB1655.DBX   75.0; //General Emergency Stop OK
      =     #EStopOK;

NETWORK
TITLE =read other unit's data

      SET   ;

// ... General Unit ----------/

      CALL FC   563 (
           ActReq                   := M    101.0,
           PLCNo                    := DB1655.DBW   14,
           SourceUnitNo             := 99,
           IsTUnit                  := FALSE,
           DstComDRec               := DB1655.GEN,
           RET_VAL                  := #wRetVal);


// ... CIP Unit ------------- /
      L     DB1651.DBD   46; // Select
      L     L#0; // Off
      ==D   ;
      JC    ELS1;
      TAK   ;
      L     DB1915.DBD   10; // CIP 1
      ==D   ;
      JC    M101;
      TAK   ;
      L     DB1925.DBD   10; // CIP 2
      ==D   ;
      JC    M102;
      TAK   ;
      L     DB1935.DBD   10; // CIP 3
      ==D   ;
      JC    M103;
      JU    ELS1;
M101: NOP   0; // Do 1
      CALL FC   563 (
           ActReq                   := M    101.0,
           PLCNo                    := 3,
           SourceUnitNo             := 91,
           IsTUnit                  := FALSE,
           DstComDRec               := DB1655.CIP,
           RET_VAL                  := #wRetVal);

      JU    FIN1;
M102: NOP   0; // Do 2
      CALL FC   563 (
           ActReq                   := M    101.0,
           PLCNo                    := 3,
           SourceUnitNo             := 92,
           IsTUnit                  := FALSE,
           DstComDRec               := DB1655.CIP,
           RET_VAL                  := #wRetVal);

      JU    FIN1;
M103: NOP   0; // Do 3
      CALL FC   563 (
           ActReq                   := M    101.0,
           PLCNo                    := 3,
           SourceUnitNo             := 93,
           IsTUnit                  := FALSE,
           DstComDRec               := DB1655.CIP,
           RET_VAL                  := #wRetVal);

      JU    FIN1;
ELS1: L     0;
      T     #iTmp;
      CALL SFC   21 (
           BVAL                     := #iTmp,
           RET_VAL                  := #iRetVal,
           BLK                      := DB1655.CIP);

FIN1: NOP   0;

NETWORK
TITLE =remote start
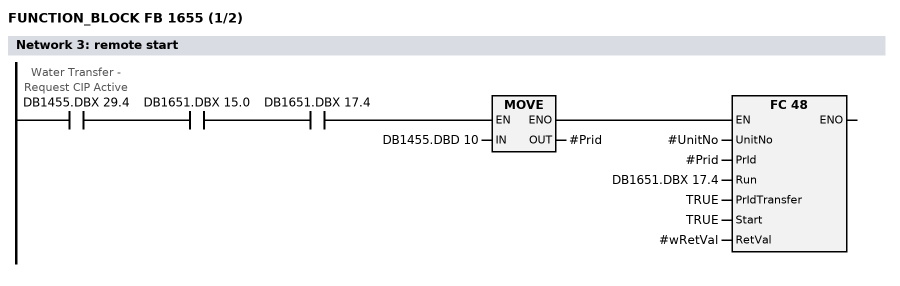

      SET   ;
      A     DB1455.DBX   29.4; // Water Transfer - Request CIP Active
      A     DB1651.DBX   15.0;
      A     DB1651.DBX   17.4;

      JCN   Strt;
      L     DB1455.DBD   10;
      T     #Prid;

      CALL FC    48 (
           UnitNo                   := #UnitNo,
           PrId                     := #Prid,
           Run                      := DB1651.DBX   17.4,
           PrIdTransfer             := TRUE,
           Start                    := TRUE,
           RetVal                   := #wRetVal);
Strt: NOP   0;
NETWORK
TITLE =external releases
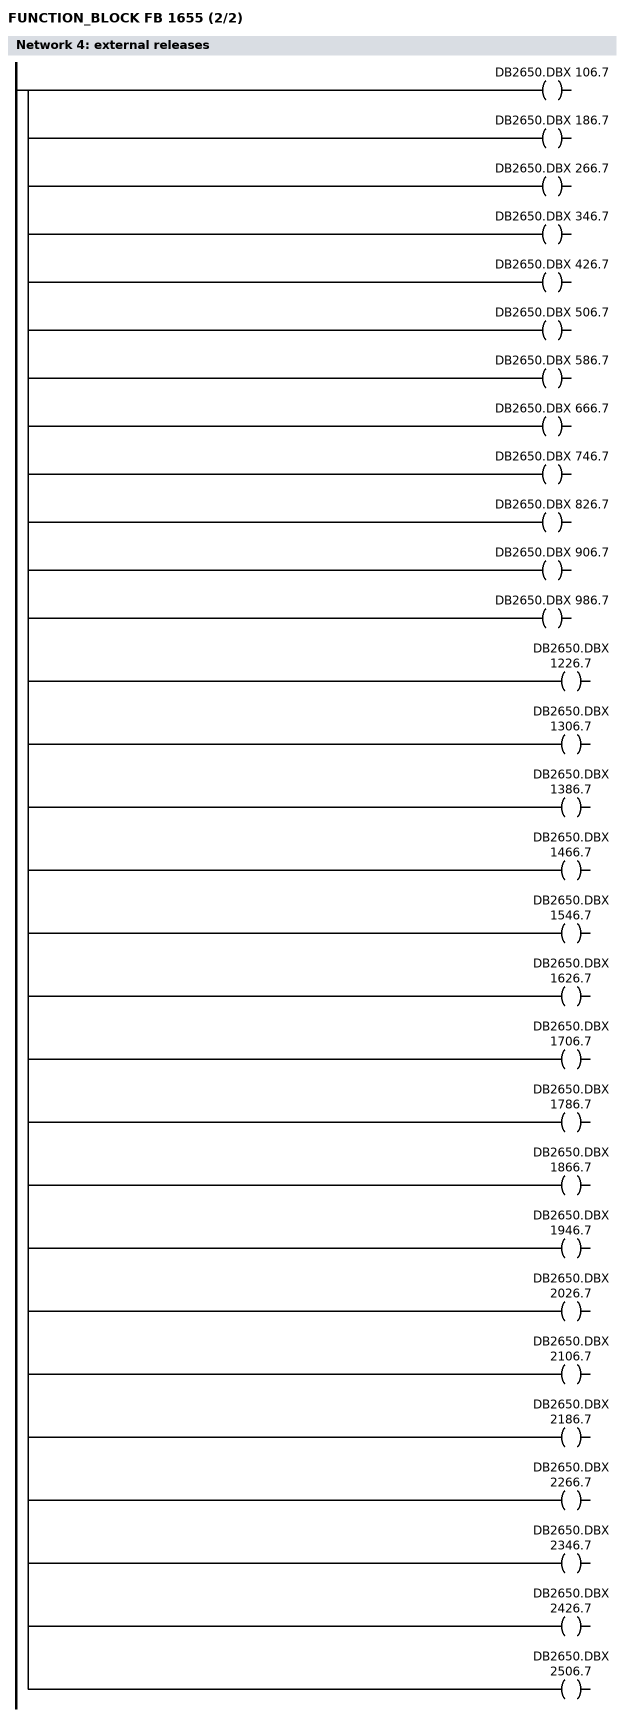

      SET   ;
      =     DB2650.DBX  106.7;
      =     DB2650.DBX  186.7;
      =     DB2650.DBX  266.7;
      =     DB2650.DBX  346.7;
      =     DB2650.DBX  426.7;
      =     DB2650.DBX  506.7;
      =     DB2650.DBX  586.7;
      =     DB2650.DBX  666.7;
      =     DB2650.DBX  746.7;
      =     DB2650.DBX  826.7;
      =     DB2650.DBX  906.7;
      =     DB2650.DBX  986.7;
      =     DB2650.DBX 1226.7;
      =     DB2650.DBX 1306.7;
      =     DB2650.DBX 1386.7;
      =     DB2650.DBX 1466.7;
      =     DB2650.DBX 1546.7;
      =     DB2650.DBX 1626.7;
      =     DB2650.DBX 1706.7;
      =     DB2650.DBX 1786.7;
      =     DB2650.DBX 1866.7;
      =     DB2650.DBX 1946.7;
      =     DB2650.DBX 2026.7;
      =     DB2650.DBX 2106.7;
      =     DB2650.DBX 2186.7;
      =     DB2650.DBX 2266.7;
      =     DB2650.DBX 2346.7;
      =     DB2650.DBX 2426.7;
      =     DB2650.DBX 2506.7;

NETWORK
TITLE =write own unit data

      SET   ;

//-- CIP Communication ---------------------------------------
      AN    DB1651.DBX   15.0;
//   AN    "U065SeqD".Seq.PO.B30       // CIP Active (Slave)  - not online
      A     #ComCIP;
      JCN   NCIP;
//Conductivity CIP Return
      L     DB1655.DBD  150;
      T     DB1651.DBD  626;

//Temperature CIP Return
      L     DB1655.DBD  146;
      T     DB1651.DBD  594;

//CIP Prerun Pump SP

      CALL FC    45 (
           SFM                      := DB1651.DBD  686,
           Indexes                  := #SFM36);


      L     0.000000e+000;
      A     #SFM36.I01;
      =     DB1655.DBX  171.7;
      JCN   pfc;
      L     DB1651.DBD  654;
pfc:  NOP   0;
      A     #SFM36.I02;
      =     DB1655.DBX  172.0;
      JCN   ppc;
      L     DB1651.DBD  670;
ppc:  NOP   0;
      A     #SFM36.I03;
      =     DB1655.DBX  171.6;
      JCN   pxc;
      L     DB1651.DBD  574;
pxc:  NOP   0;
      T     DB1655.DBD  182;

//CIP Return
      L     DB1651.DBD  558;
      T     DB1655.DBD  186;
      L     DB1655.DBD  138;
      T     DB1651.DBD  562;

//CIP Prerun
      L     DB1651.DBD  542;
      T     DB1655.DBD  190;
      L     DB1655.DBD  142;
      T     DB1651.DBD  546;

// Write Own Data to CIP
      L     DB1655.DBD   10;
      T     DB1655.DBD  154;

      L     DB1655.DBW   14;
      T     DB1655.DBW  158;

      L     DB1655.DBW   16;
      T     DB1655.DBW  160;

      L     DB1655.DBW   18;
      T     DB1655.DBW  162;

      L     DB1655.DBW   20;
      T     DB1655.DBW  164;

      L     DB1655.DBW   22;
      T     DB1655.DBW  166;

      A     DB1655.DBX   24.0;
      =     DB1655.DBX  168.0;

      A     DB1655.DBX   24.1;
      =     DB1655.DBX  168.1;

      A     DB1655.DBX   24.2;
      =     DB1655.DBX  168.2;

      A     DB1655.DBX   24.3;
      =     DB1655.DBX  168.3;

      A     DB1655.DBX   24.4;
      =     DB1655.DBX  168.4;

      A     DB1655.DBX   24.5;
      =     DB1655.DBX  168.5;

      A     DB1655.DBX   24.6;
      =     DB1655.DBX  168.6;

      A     DB1655.DBX   24.7;
      =     DB1655.DBX  168.7;

// Copy Data to CIP
      CALL SFC   20 (
           SRCBLK                   := DB1655.ToCIP,
           RET_VAL                  := #iRetVal,
           DSTBLK                   := DB1655.ToCIP);

NCIP: NOP   0;

//Empty Signal
//A     "U065SpID".SpI.Sig //!!!! Insert correct Empty Signal !!!
      CLR   ;
      =     DB1655.DBX   26.5;

//Full Signal
//A     "U065SpID".SpI.Sig //!!!! Insert correct Full Signal !!!
      CLR   ;
      =     DB1655.DBX   26.2;

//CIP Program Selected
      A     #CIP;
      =     DB1655.DBX   27.1;

// Emergency Stop
      A     #EStopOK; //If needed add or replace with own SpI
      =     DB1655.DBX   27.0; //Emergency Stop OK


NETWORK
TITLE =Signals to Filler / Mixer

// Watchdog
      A     M    100.7;
      =     Q    197.7;
      =     Q    173.7;
      =     Q    199.6;
      =     Q    345.7;

// GOA Panel
      A     I    194.0;
      =     DB5050.DBX 2028.2;

      A     I    194.1;
      =     DB5050.DBX 2188.2;

      A     I    194.2;
      =     DB5050.DBX 2348.2;

      CLR   ;

      L     DB2653.DBD  146;
      T     QD   356;
END_FUNCTION_BLOCK

FUNCTION_BLOCK FB 1659
TITLE =U065: Packaging Plant 5
AUTHOR : Woermann
FAMILY : BOTEC_F1
NAME : Sim
VERSION : 0.1


VAR_TEMP
  CIP : BOOL ;	//CIP active
  xTmp : BOOL ;	//Temporary BOOL (free for general use)
  iTmp : INT ;	//Temporary INT (free for general use)
  rTmp : REAL ;	//Temporary REAL (free for general use)
  UnitNo : INT ;	//Unit Number
END_VAR
BEGIN
NETWORK
TITLE =General

      SET   ;
// get unit number ----------------------------------------------------------
      L     DB1650.DBW    0;
      T     #UnitNo;

// CIP ----------------------------------------------------------------------
      L     DB1651.DBD   54;
      L     0;
      <D    ;
      =     #CIP;

NETWORK
TITLE =Actuator

      A     DB1651.DBX   17.3;
      =     DB2650.DBX  105.3;
      =     DB2650.DBX  185.3;
      =     DB2650.DBX  265.3;
      =     DB2650.DBX  345.3;
      =     DB2650.DBX  425.3;
      =     DB2650.DBX  505.3;
      =     DB2650.DBX  585.3;
      =     DB2650.DBX  665.3;
      =     DB2650.DBX  745.3;
      =     DB2650.DBX  825.3;
      =     DB2650.DBX  905.3;
      =     DB2650.DBX  985.3;
      =     DB2650.DBX 1225.3;
      =     DB2650.DBX 1305.3;
      =     DB2650.DBX 1385.3;
      =     DB2650.DBX 1465.3;
      =     DB2650.DBX 1545.3;
      =     DB2650.DBX 1625.3;
      =     DB2650.DBX 1705.3;
      =     DB2650.DBX 1785.3;
      =     DB2650.DBX 1865.3;
      =     DB2650.DBX 1945.3;
      =     DB2650.DBX 2025.3;
      =     DB2650.DBX 2105.3;
      =     DB2650.DBX 2185.3;
      =     DB2650.DBX 2265.3;
      =     DB2650.DBX 2345.3;
      =     DB2650.DBX 2425.3;
      =     DB2650.DBX 2505.3;
      =     DB2650.DBX 2585.3;
      =     DB2650.DBX 2665.3;
      =     DB2650.DBX 2745.3;
      =     DB2650.DBX 2825.3;
      =     DB2650.DBX 2905.3;
      =     DB2650.DBX 2985.3;
      =     DB2650.DBX 3065.3;
      =     DB2650.DBX 3145.3;
      =     DB2650.DBX 3225.3;
      =     DB2650.DBX 3305.3;
      =     DB2650.DBX 3385.3;
      =     DB2650.DBX 3465.3;
      =     DB2650.DBX 3545.3;
      =     DB2650.DBX 3625.3;
      =     DB2650.DBX 3705.3;
      =     DB2650.DBX 3785.3;
      =     DB2650.DBX 3865.3;
      =     DB2650.DBX 3945.3;
      =     DB2650.DBX 4025.3;
      =     DB2650.DBX 4105.3;
      =     DB2650.DBX 4185.3;
      =     DB2650.DBX 4265.3;
      =     DB2650.DBX 4345.3;
      =     DB2650.DBX 4425.3;
      =     DB2650.DBX 4505.3;
      =     DB2650.DBX 4585.3;
      =     DB2650.DBX 4665.3;
      =     DB2650.DBX 4745.3;
      =     DB2650.DBX 4825.3;
      =     DB2650.DBX 4905.3;
      =     DB2650.DBX 4985.3;
      =     DB2650.DBX 5065.3;
      =     DB2650.DBX 5145.3;
      =     DB2650.DBX 5225.3;
      =     DB2650.DBX 5385.3;
      =     DB2650.DBX 5465.3;
      =     DB2650.DBX 5545.3;
      =     DB2650.DBX 5625.3;
      =     DB2650.DBX 5705.3;
      =     DB2650.DBX 5785.3;

NETWORK
TITLE =Special Input

      A     DB1651.DBX   17.3;
      =     DB2651.DBX  141.3;
      =     DB2651.DBX  201.3;
      =     DB2651.DBX  261.3;
      =     DB2651.DBX  321.3;
      =     DB2651.DBX  381.3;
      =     DB2651.DBX  441.3;
      =     DB2651.DBX  501.3;
      =     DB2651.DBX  561.3;
      =     DB2651.DBX  621.3;
      =     DB2651.DBX  681.3;
      =     DB2651.DBX 1881.3;
      =     DB2651.DBX 1941.3;
      =     DB2651.DBX 2001.3;
      =     DB2651.DBX 2061.3;
      =     DB2651.DBX 2121.3;
      =     DB2651.DBX 2181.3;
      =     DB2651.DBX 2421.3;
      =     DB2651.DBX 2481.3;
      =     DB2651.DBX 2541.3;
      =     DB2651.DBX 2721.3;
      =     DB2651.DBX 2781.3;
      =     DB2651.DBX 2841.3;
      =     DB2651.DBX 2901.3;
      =     DB2651.DBX 2961.3;
      =     DB2651.DBX 3021.3;
      =     DB2651.DBX 3081.3;
      =     DB2651.DBX 3141.3;
      =     DB2651.DBX 3201.3;
      =     DB2651.DBX 3261.3;
      =     DB2651.DBX 3321.3;
      =     DB2651.DBX 3381.3;
      =     DB2651.DBX 3441.3;

NETWORK
TITLE =Counter

      A     DB1651.DBX   17.3;
      A     M    101.0;


      CLR   ;
NETWORK
TITLE =Analog Input

      A     DB1651.DBX   17.3;
      =     DB2653.DBX  141.3;
      =     DB2653.DBX  261.3;
      =     DB2653.DBX  381.3;
      =     DB2653.DBX  501.3;
      =     DB2653.DBX  621.3;
      =     DB2653.DBX  741.3;

NETWORK
TITLE =Universal Value

      A     DB1651.DBX   17.3;
//      =     "U065UnVD".unv001.Sim;
//      =     "U065UnVD".unv002.Sim;
//      =     "U065UnVD".unv003.Sim;
//      =     "U065UnVD".unv004.Sim;

NETWORK
TITLE =PID

      A     DB1651.DBX   17.3;

NETWORK
TITLE =Message

      A     DB1651.DBX   17.3;
//      =     "U065MsgD".msg001.Sim;
//      =     "U065MsgD".msg002.Sim;
//      =     "U065MsgD".msg003.Sim;

NETWORK
TITLE =VLT

      A     DB1651.DBX   17.3;

END_FUNCTION_BLOCK

FUNCTION_BLOCK FB 1675
TITLE =U067: Packaging Plant 7
FAMILY : BOTEC_F1
NAME : Comm
VERSION : 0.1


VAR_TEMP
  iRetVal : INT ;	//return value as integer
  wRetVal : WORD ;	//return value as word
  Run : BOOL ;	//Unit in "RUN" mode
  EStopOK : BOOL ;	//Emergency Stop OK
  CIP : BOOL ;	//CIP Program Selected
  ComCIP : BOOL ;	//Communication with CIP Active
  xTmp : BOOL ;	//Temporary BOOL (free for general use)
  iTmp : INT ;	//Temporary INT (free for general use)
  rTmp : REAL ;	//Temporary REAL (free for general use)
  dTmp : DINT ;	//Temporary DINT (free for general use)
  UnitNo : INT ;	//Unit Number
  EquipmentID : INT ;	//Equipment ID
  Prid : DINT ;	//Process ID
  SFM36 : STRUCT 	// CIP Pump Mode
   I00 : BOOL ;	// Off
   I01 : BOOL ;	// Flow
   I02 : BOOL ;	// Pressure
   I03 : BOOL ;	// Fix Speed
   I04 : BOOL ;
   I05 : BOOL ;
   I06 : BOOL ;
   I07 : BOOL ;
   I08 : BOOL ;
   I09 : BOOL ;
   I10 : BOOL ;
   I11 : BOOL ;
   I12 : BOOL ;
   I13 : BOOL ;
   I14 : BOOL ;
   I15 : BOOL ;
   I16 : BOOL ;
   I17 : BOOL ;
   I18 : BOOL ;
   I19 : BOOL ;
   I20 : BOOL ;
   I21 : BOOL ;
   I22 : BOOL ;
   I23 : BOOL ;
   I24 : BOOL ;
   I25 : BOOL ;
   I26 : BOOL ;
   I27 : BOOL ;
   I28 : BOOL ;
   I29 : BOOL ;
   I30 : BOOL ;
   I31 : BOOL ;
  END_STRUCT ;
END_VAR
BEGIN
NETWORK
TITLE =general

      SET   ;

// unit & equipment number ---------------------------------------------------
      L     DB1670.DBW    0;
      T     #UnitNo;

      L     DB1675.DBW   14;
      L     1000;
      *I    ;
      L     #UnitNo;
      +I    ;
      T     #EquipmentID;

// CIP ----------------------------------------------------------------------
      L     DB1675.DBW   18;
      L     0;
      <I    ;
      =     #CIP;

// Communicating Units-------------------------------------------------------
      L     DB1675.DBD   10;
      L     DB1675.DBD  106;
      ==D   ;
      =     #ComCIP;

// emergency OK -------------------------------------------------------------
      A     DB1675.DBX   75.0; //General Emergency Stop OK
      =     #EStopOK;

NETWORK
TITLE =read other unit's data

      SET   ;

// ... General Unit ----------/

      CALL FC   563 (
           ActReq                   := M    101.0,
           PLCNo                    := DB1675.DBW   14,
           SourceUnitNo             := 99,
           IsTUnit                  := FALSE,
           DstComDRec               := DB1675.GEN,
           RET_VAL                  := #wRetVal);


// ... CIP Unit ------------- /
      L     DB1671.DBD   46; // Select
      L     L#0; // Off
      ==D   ;
      JC    ELS1;
      TAK   ;
      L     DB1915.DBD   10; // CIP 1
      ==D   ;
      JC    M101;
      TAK   ;
      L     DB1925.DBD   10; // CIP 2
      ==D   ;
      JC    M102;
      TAK   ;
      L     DB1935.DBD   10; // CIP 3
      ==D   ;
      JC    M103;
      JU    ELS1;
M101: NOP   0; // Do 1
      CALL FC   563 (
           ActReq                   := M    101.0,
           PLCNo                    := 3,
           SourceUnitNo             := 91,
           IsTUnit                  := FALSE,
           DstComDRec               := DB1675.CIP,
           RET_VAL                  := #wRetVal);

      JU    FIN1;
M102: NOP   0; // Do 2
      CALL FC   563 (
           ActReq                   := M    101.0,
           PLCNo                    := 3,
           SourceUnitNo             := 92,
           IsTUnit                  := FALSE,
           DstComDRec               := DB1675.CIP,
           RET_VAL                  := #wRetVal);

      JU    FIN1;
M103: NOP   0; // Do 3
      CALL FC   563 (
           ActReq                   := M    101.0,
           PLCNo                    := 3,
           SourceUnitNo             := 93,
           IsTUnit                  := FALSE,
           DstComDRec               := DB1675.CIP,
           RET_VAL                  := #wRetVal);

      JU    FIN1;
ELS1: L     0;
      T     #iTmp;
      CALL SFC   21 (
           BVAL                     := #iTmp,
           RET_VAL                  := #iRetVal,
           BLK                      := DB1675.CIP);

FIN1: NOP   0;

NETWORK
TITLE =remote start
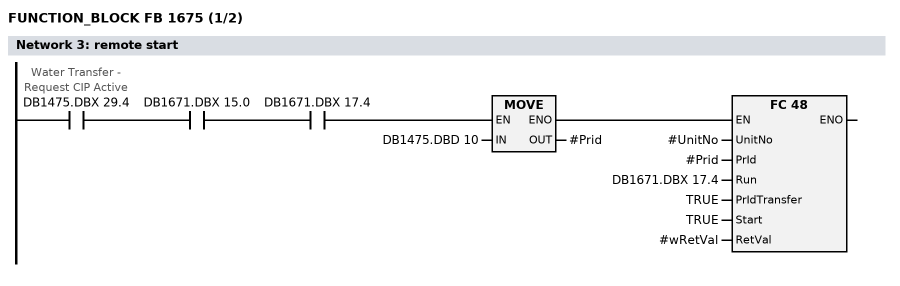

      SET   ;
      A     DB1475.DBX   29.4; // Water Transfer - Request CIP Active
      A     DB1671.DBX   15.0;
      A     DB1671.DBX   17.4;

      JCN   Strt;
      L     DB1475.DBD   10;
      T     #Prid;

      CALL FC    48 (
           UnitNo                   := #UnitNo,
           PrId                     := #Prid,
           Run                      := DB1671.DBX   17.4,
           PrIdTransfer             := TRUE,
           Start                    := TRUE,
           RetVal                   := #wRetVal);
Strt: NOP   0;
NETWORK
TITLE =external releases
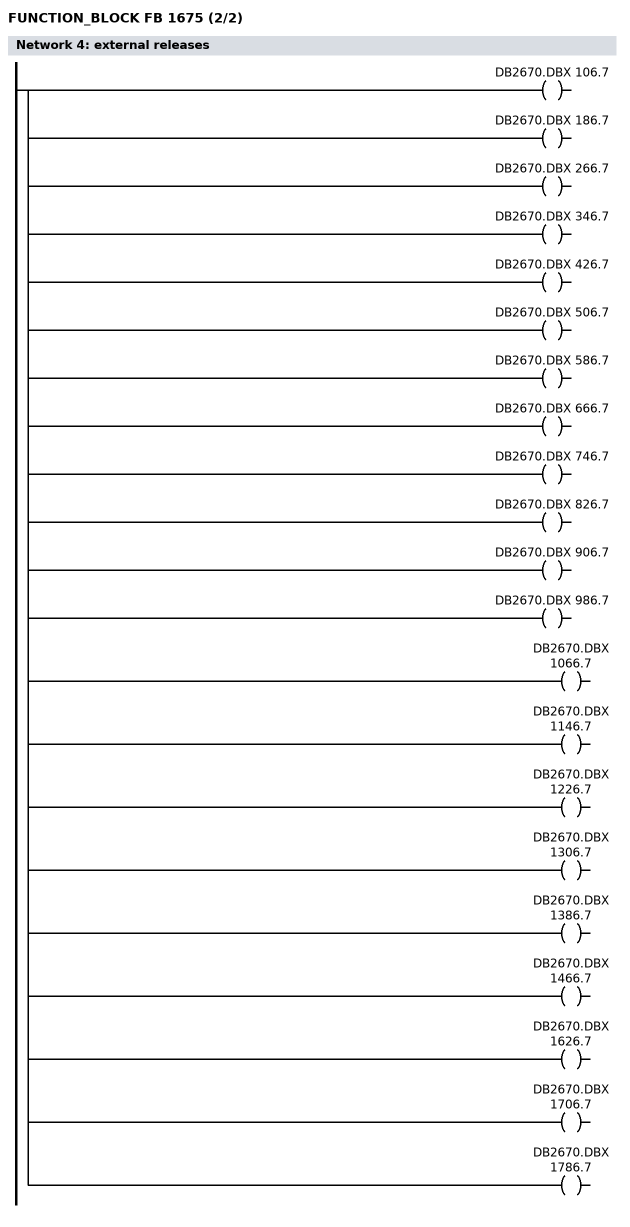

      SET   ;
      =     DB2670.DBX  106.7;
      =     DB2670.DBX  186.7;
      =     DB2670.DBX  266.7;
      =     DB2670.DBX  346.7;
      =     DB2670.DBX  426.7;
      =     DB2670.DBX  506.7;
      =     DB2670.DBX  586.7;
      =     DB2670.DBX  666.7;
      =     DB2670.DBX  746.7;
      =     DB2670.DBX  826.7;
      =     DB2670.DBX  906.7;
      =     DB2670.DBX  986.7;
      =     DB2670.DBX 1066.7;
      =     DB2670.DBX 1146.7;
      =     DB2670.DBX 1226.7;
      =     DB2670.DBX 1306.7;
      =     DB2670.DBX 1386.7;
      =     DB2670.DBX 1466.7;
      =     DB2670.DBX 1626.7;
      =     DB2670.DBX 1706.7;
      =     DB2670.DBX 1786.7;
NETWORK
TITLE =write own unit data

      SET   ;

//-- CIP Communication ---------------------------------------
      AN    DB1671.DBX   15.0;
      AN    DB1671.DBX 1233.6; // CIP Active (Slave)
      A     #ComCIP;
      JCN   NCIP;
//Conductivity CIP Return
      L     DB1675.DBD  150;
      T     DB1671.DBD  626;

//Temperature CIP Return
      L     DB1675.DBD  146;
      T     DB1671.DBD  594;

//CIP Prerun Pump SP

      CALL FC    45 (
           SFM                      := DB1671.DBD  686,
           Indexes                  := #SFM36);


      L     0.000000e+000;
      A     #SFM36.I01;
      =     DB1675.DBX  171.7;
      JCN   pfc;
      L     DB1671.DBD  654;
pfc:  NOP   0;
      A     #SFM36.I02;
      =     DB1675.DBX  172.0;
      JCN   ppc;
      L     DB1671.DBD  670;
ppc:  NOP   0;
      A     #SFM36.I03;
      =     DB1675.DBX  171.6;
      JCN   pxc;
      L     DB1671.DBD  574;
pxc:  NOP   0;
      T     DB1675.DBD  182;

//CIP Return
      L     DB1671.DBD  558;
      T     DB1675.DBD  186;
      L     DB1675.DBD  138;
      T     DB1671.DBD  562;

//CIP Prerun
      L     DB1671.DBD  542;
      T     DB1675.DBD  190;
      L     DB1675.DBD  142;
      T     DB1671.DBD  546;

// Write Own Data to CIP
      L     DB1675.DBD   10;
      T     DB1675.DBD  154;

      L     DB1675.DBW   14;
      T     DB1675.DBW  158;

      L     DB1675.DBW   16;
      T     DB1675.DBW  160;

      L     DB1675.DBW   18;
      T     DB1675.DBW  162;

      L     DB1675.DBW   20;
      T     DB1675.DBW  164;

      L     DB1675.DBW   22;
      T     DB1675.DBW  166;

      A     DB1675.DBX   24.0;
      =     DB1675.DBX  168.0;

      A     DB1675.DBX   24.1;
      =     DB1675.DBX  168.1;

      A     DB1675.DBX   24.2;
      =     DB1675.DBX  168.2;

      A     DB1675.DBX   24.3;
      =     DB1675.DBX  168.3;

      A     DB1675.DBX   24.4;
      =     DB1675.DBX  168.4;

      A     DB1675.DBX   24.5;
      =     DB1675.DBX  168.5;

      A     DB1675.DBX   24.6;
      =     DB1675.DBX  168.6;

      A     DB1675.DBX   24.7;
      =     DB1675.DBX  168.7;

// Copy Data to CIP
      CALL SFC   20 (
           SRCBLK                   := DB1675.ToCIP,
           RET_VAL                  := #iRetVal,
           DSTBLK                   := DB1675.ToCIP);

NCIP: NOP   0;

//Empty Signal
//A     "U067SpID".SpI.Sig //!!!! Insert correct Empty Signal !!!
      CLR   ;
      =     DB1675.DBX   26.5;

//Full Signal
//A     "U067SpID".SpI.Sig //!!!! Insert correct Full Signal !!!
      CLR   ;
      =     DB1675.DBX   26.2;

//CIP Program Selected
      A     #CIP;
      =     DB1675.DBX   27.1;

// Emergency Stop
      A     #EStopOK; //If needed add or replace with own SpI
      =     DB1675.DBX   27.0; //Emergency Stop OK


NETWORK
TITLE = read from other unit data

//    A     "U107SpID".GOA_701.Sig
      A     I     26.0;
      =     DB5070.DBX 1788.2;

//    A     "U107SpID".GOA_702.Sig
      A     I     26.1;
      =     DB5070.DBX 1868.2;

//    A     "U067SpID".GOA_703.Sig
      A     I     26.2;
      =     DB5070.DBX 1948.2;





      CLR   ;
END_FUNCTION_BLOCK

FUNCTION_BLOCK FB 1679
TITLE =U067: Packaging Plant 7
AUTHOR : Woermann
FAMILY : BOTEC_F1
NAME : Sim
VERSION : 0.1


VAR_TEMP
  CIP : BOOL ;	//CIP active
  xTmp : BOOL ;	//Temporary BOOL (free for general use)
  iTmp : INT ;	//Temporary INT (free for general use)
  rTmp : REAL ;	//Temporary REAL (free for general use)
  UnitNo : INT ;	//Unit Number
END_VAR
BEGIN
NETWORK
TITLE =General

      SET   ;
// get unit number ----------------------------------------------------------
      L     DB1670.DBW    0;
      T     #UnitNo;

// CIP ----------------------------------------------------------------------
      L     DB1671.DBD   54;
      L     0;
      <D    ;
      =     #CIP;

NETWORK
TITLE =Actuator

      A     DB1671.DBX   17.3;
      =     DB2670.DBX  105.3;
      =     DB2670.DBX  185.3;
      =     DB2670.DBX  265.3;
      =     DB2670.DBX  345.3;
      =     DB2670.DBX  425.3;
      =     DB2670.DBX  505.3;
      =     DB2670.DBX  585.3;
      =     DB2670.DBX  665.3;
      =     DB2670.DBX  745.3;
      =     DB2670.DBX  825.3;
      =     DB2670.DBX  905.3;
      =     DB2670.DBX  985.3;
      =     DB2670.DBX 1065.3;
      =     DB2670.DBX 1145.3;
      =     DB2670.DBX 1225.3;
      =     DB2670.DBX 1305.3;
      =     DB2670.DBX 1385.3;
      =     DB2670.DBX 1465.3;
      =     DB2670.DBX 1625.3;
      =     DB2670.DBX 1705.3;
      =     DB2670.DBX 1785.3;

NETWORK
TITLE =Special Input

      A     DB1671.DBX   17.3;
      CLR   ;
      =     DB2671.DBX  141.3;
      =     DB2671.DBX  201.3;
      =     DB2671.DBX  261.3;
      =     DB2671.DBX  321.3;
      =     DB2671.DBX  381.3;
      =     DB2671.DBX  441.3;
      =     DB2671.DBX  561.3;
      =     DB2671.DBX  681.3;
      =     DB2671.DBX  801.3;
      =     DB2671.DBX  861.3;
      =     DB2671.DBX  921.3;




NETWORK
TITLE =Counter

      A     DB1671.DBX   17.3;
      A     M    101.0;


      CLR   ;
NETWORK
TITLE =Analog Input

      A     DB1671.DBX   17.3;

NETWORK
TITLE =Universal Value

      A     DB1671.DBX   17.3;
//      =     "U067UnVD".unv001.Sim;
//      =     "U067UnVD".unv002.Sim;
//      =     "U067UnVD".unv003.Sim;
//      =     "U067UnVD".unv004.Sim;

NETWORK
TITLE =PID

      A     DB1671.DBX   17.3;

NETWORK
TITLE =Message

      A     DB1671.DBX   17.3;
//      =     "U067MsgD".msg001.Sim;
//      =     "U067MsgD".msg002.Sim;
//      =     "U067MsgD".msg003.Sim;

NETWORK
TITLE =VLT

      A     DB1671.DBX   17.3;

END_FUNCTION_BLOCK

FUNCTION_BLOCK FB 1685
TITLE =U068: Packaging Plant 8
FAMILY : BOTEC_F1
NAME : Comm
VERSION : 0.1


VAR_TEMP
  iRetVal : INT ;	//return value as integer
  wRetVal : WORD ;	//return value as word
  Run : BOOL ;	//Unit in "RUN" mode
  EStopOK : BOOL ;	//Emergency Stop OK
  CIP : BOOL ;	//CIP Program Selected
  ComCIP : BOOL ;	//Communication with CIP Active
  xTmp : BOOL ;	//Temporary BOOL (free for general use)
  iTmp : INT ;	//Temporary INT (free for general use)
  rTmp : REAL ;	//Temporary REAL (free for general use)
  dTmp : DINT ;	//Temporary DINT (free for general use)
  UnitNo : INT ;	//Unit Number
  EquipmentID : INT ;	//Equipment ID
  Prid : DINT ;	//Process ID
  SFM36 : STRUCT 	// CIP Pump Mode
   I00 : BOOL ;	// Off
   I01 : BOOL ;	// Flow
   I02 : BOOL ;	// Pressure
   I03 : BOOL ;	// Fix Speed
   I04 : BOOL ;
   I05 : BOOL ;
   I06 : BOOL ;
   I07 : BOOL ;
   I08 : BOOL ;
   I09 : BOOL ;
   I10 : BOOL ;
   I11 : BOOL ;
   I12 : BOOL ;
   I13 : BOOL ;
   I14 : BOOL ;
   I15 : BOOL ;
   I16 : BOOL ;
   I17 : BOOL ;
   I18 : BOOL ;
   I19 : BOOL ;
   I20 : BOOL ;
   I21 : BOOL ;
   I22 : BOOL ;
   I23 : BOOL ;
   I24 : BOOL ;
   I25 : BOOL ;
   I26 : BOOL ;
   I27 : BOOL ;
   I28 : BOOL ;
   I29 : BOOL ;
   I30 : BOOL ;
   I31 : BOOL ;
  END_STRUCT ;
END_VAR
BEGIN
NETWORK
TITLE =general

      SET   ;

// unit & equipment number ---------------------------------------------------
      L     DB1680.DBW    0;
      T     #UnitNo;

      L     DB1685.DBW   14;
      L     1000;
      *I    ;
      L     #UnitNo;
      +I    ;
      T     #EquipmentID;

// CIP ----------------------------------------------------------------------
      L     DB1685.DBW   18;
      L     0;
      <I    ;
      =     #CIP;

// Communicating Units-------------------------------------------------------
      L     DB1685.DBD   10;
      L     DB1685.DBD  106;
      ==D   ;
      =     #ComCIP;

// emergency OK -------------------------------------------------------------
      A     DB1685.DBX   75.0; //General Emergency Stop OK
      =     #EStopOK;

NETWORK
TITLE =read other unit's data

      SET   ;

// ... General Unit ----------/

      CALL FC   563 (
           ActReq                   := M    101.0,
           PLCNo                    := DB1685.DBW   14,
           SourceUnitNo             := 99,
           IsTUnit                  := FALSE,
           DstComDRec               := DB1685.GEN,
           RET_VAL                  := #wRetVal);

NETWORK
TITLE =remote start

      SET   ;
// !!! insert correct condition of unit start !!!
      A     DB1681.DBX   15.0;
      A     DB1681.DBX   17.4;
      CLR   ;
      JCN   Strt;
      L     DB1685.DBD   10;
//L        L#-1;                            // Prid negative to start on its own
      T     #Prid;

      CALL FC    48 (
           UnitNo                   := #UnitNo,
           PrId                     := #Prid,
           Run                      := DB1681.DBX   17.4,
           PrIdTransfer             := TRUE,
           Start                    := TRUE,
           RetVal                   := #wRetVal);
Strt: NOP   0;
NETWORK
TITLE =external releases

      SET   ;
      =     DB2680.DBX  106.7;
      =     DB2680.DBX  186.7;
      =     DB2680.DBX  266.7;
      =     DB2680.DBX  346.7;
      =     DB2680.DBX  426.7;
      =     DB2680.DBX  506.7;
      =     DB2680.DBX  586.7;
      =     DB2680.DBX  666.7;
      =     DB2680.DBX  746.7;
      =     DB2680.DBX  826.7;
      =     DB2680.DBX 1626.7;
      =     DB2680.DBX 1706.7;
      =     DB2680.DBX 1786.7;
NETWORK
TITLE =write own unit data

      SET   ;

//-- CIP Communication ---------------------------------------
      AN    DB1681.DBX   15.0;
//      AN "U068SeqD".Seq.PO.B30 // CIP Active (Slave)
      A     #ComCIP;
      JCN   NCIP;
//Conductivity CIP Return
      L     DB1685.DBD  150;
      T     DB1681.DBD  626;

//Temperature CIP Return
      L     DB1685.DBD  146;
      T     DB1681.DBD  594;

//CIP Prerun Pump SP

      CALL FC    45 (
           SFM                      := DB1681.DBD  686,
           Indexes                  := #SFM36);


      L     0.000000e+000;
      A     #SFM36.I01;
      =     DB1685.DBX  171.7;
      JCN   pfc;
      L     DB1681.DBD  654;
pfc:  NOP   0;
      A     #SFM36.I02;
      =     DB1685.DBX  172.0;
      JCN   ppc;
      L     DB1681.DBD  670;
ppc:  NOP   0;
      A     #SFM36.I03;
      =     DB1685.DBX  171.6;
      JCN   pxc;
      L     DB1681.DBD  574;
pxc:  NOP   0;
      T     DB1685.DBD  182;

//CIP Return
      L     DB1681.DBD  558;
      T     DB1685.DBD  186;
      L     DB1685.DBD  138;
      T     DB1681.DBD  562;

//CIP Prerun
      L     DB1681.DBD  542;
      T     DB1685.DBD  190;
      L     DB1685.DBD  142;
      T     DB1681.DBD  546;

// Write Own Data to CIP
      L     DB1685.DBD   10;
      T     DB1685.DBD  154;

      L     DB1685.DBW   14;
      T     DB1685.DBW  158;

      L     DB1685.DBW   16;
      T     DB1685.DBW  160;

      L     DB1685.DBW   18;
      T     DB1685.DBW  162;

      L     DB1685.DBW   20;
      T     DB1685.DBW  164;

      L     DB1685.DBW   22;
      T     DB1685.DBW  166;

      A     DB1685.DBX   24.0;
      =     DB1685.DBX  168.0;

      A     DB1685.DBX   24.1;
      =     DB1685.DBX  168.1;

      A     DB1685.DBX   24.2;
      =     DB1685.DBX  168.2;

      A     DB1685.DBX   24.3;
      =     DB1685.DBX  168.3;

      A     DB1685.DBX   24.4;
      =     DB1685.DBX  168.4;

      A     DB1685.DBX   24.5;
      =     DB1685.DBX  168.5;

      A     DB1685.DBX   24.6;
      =     DB1685.DBX  168.6;

      A     DB1685.DBX   24.7;
      =     DB1685.DBX  168.7;

// Copy Data to CIP
      CALL SFC   20 (
           SRCBLK                   := DB1685.ToCIP,
           RET_VAL                  := #iRetVal,
           DSTBLK                   := DB1685.ToCIP);

NCIP: NOP   0;

//Empty Signal
//A     "U068SpID".SpI.Sig //!!!! Insert correct Empty Signal !!!
      CLR   ;
      =     DB1685.DBX   26.5;

//Full Signal
//A     "U068SpID".SpI.Sig //!!!! Insert correct Full Signal !!!
      CLR   ;
      =     DB1685.DBX   26.2;

//CIP Program Selected
      A     #CIP;
      =     DB1685.DBX   27.1;

// Emergency Stop
      A     #EStopOK; //If needed add or replace with own SpI
      =     DB1685.DBX   27.0; //Emergency Stop OK


NETWORK
TITLE = read from other unit data



END_FUNCTION_BLOCK

FUNCTION_BLOCK FB 1689
TITLE =U068: Packaging Plant 8
AUTHOR : Woermann
FAMILY : BOTEC_F1
NAME : Sim
VERSION : 0.1


VAR_TEMP
  CIP : BOOL ;	//CIP active
  xTmp : BOOL ;	//Temporary BOOL (free for general use)
  iTmp : INT ;	//Temporary INT (free for general use)
  rTmp : REAL ;	//Temporary REAL (free for general use)
  UnitNo : INT ;	//Unit Number
END_VAR
BEGIN
NETWORK
TITLE =General

      SET   ;
// get unit number ----------------------------------------------------------
      L     DB1680.DBW    0;
      T     #UnitNo;

// CIP ----------------------------------------------------------------------
      L     DB1681.DBD   54;
      L     0;
      <D    ;
      =     #CIP;

NETWORK
TITLE =Actuator

      A     DB1681.DBX   17.3;
      =     DB2680.DBX  105.3;
      =     DB2680.DBX  185.3;
      =     DB2680.DBX  265.3;
      =     DB2680.DBX  345.3;
      =     DB2680.DBX  425.3;
      =     DB2680.DBX  505.3;
      =     DB2680.DBX  585.3;
      =     DB2680.DBX  665.3;
      =     DB2680.DBX  745.3;
      =     DB2680.DBX  825.3;
      =     DB2680.DBX 1625.3;
      =     DB2680.DBX 1705.3;
      =     DB2680.DBX 1785.3;

NETWORK
TITLE =Special Input

      A     DB1681.DBX   17.3;
      =     DB2681.DBX  141.3;
      =     DB2681.DBX  201.3;
      =     DB2681.DBX  681.3;
      =     DB2681.DBX 1461.3;
      =     DB2681.DBX 1521.3;
      =     DB2681.DBX 1581.3;
      =     DB2681.DBX 1641.3;
      =     DB2681.DBX 1701.3;

NETWORK
TITLE =Counter

      A     DB1681.DBX   17.3;
      A     M    101.0;


      CLR   ;
NETWORK
TITLE =Analog Input

      A     DB1681.DBX   17.3;

NETWORK
TITLE =Universal Value

      A     DB1681.DBX   17.3;
//      =     "U068UnVD".unv001.Sim;
//      =     "U068UnVD".unv002.Sim;
//      =     "U068UnVD".unv003.Sim;
//      =     "U068UnVD".unv004.Sim;

NETWORK
TITLE =PID

      A     DB1681.DBX   17.3;

NETWORK
TITLE =Message

      A     DB1681.DBX   17.3;
//      =     "U068MsgD".msg001.Sim;
//      =     "U068MsgD".msg002.Sim;
//      =     "U068MsgD".msg003.Sim;

NETWORK
TITLE =VLT

      A     DB1681.DBX   17.3;

END_FUNCTION_BLOCK

FUNCTION_BLOCK FB 1695
TITLE =U069: Packaging Plant 9
FAMILY : BOTEC_F1
NAME : Comm
VERSION : 0.1


VAR_TEMP
  iRetVal : INT ;	//return value as integer
  wRetVal : WORD ;	//return value as word
  Run : BOOL ;	//Unit in "RUN" mode
  EStopOK : BOOL ;	//Emergency Stop OK
  CIP : BOOL ;	//CIP Program Selected
  ComCIP : BOOL ;	//Communication with CIP Active
  xTmp : BOOL ;	//Temporary BOOL (free for general use)
  iTmp : INT ;	//Temporary INT (free for general use)
  rTmp : REAL ;	//Temporary REAL (free for general use)
  dTmp : DINT ;	//Temporary DINT (free for general use)
  UnitNo : INT ;	//Unit Number
  EquipmentID : INT ;	//Equipment ID
  Prid : DINT ;	//Process ID
  SFM36 : STRUCT 	// CIP Pump Mode
   I00 : BOOL ;	// Off
   I01 : BOOL ;	// Flow
   I02 : BOOL ;	// Pressure
   I03 : BOOL ;	// Fix Speed
   I04 : BOOL ;
   I05 : BOOL ;
   I06 : BOOL ;
   I07 : BOOL ;
   I08 : BOOL ;
   I09 : BOOL ;
   I10 : BOOL ;
   I11 : BOOL ;
   I12 : BOOL ;
   I13 : BOOL ;
   I14 : BOOL ;
   I15 : BOOL ;
   I16 : BOOL ;
   I17 : BOOL ;
   I18 : BOOL ;
   I19 : BOOL ;
   I20 : BOOL ;
   I21 : BOOL ;
   I22 : BOOL ;
   I23 : BOOL ;
   I24 : BOOL ;
   I25 : BOOL ;
   I26 : BOOL ;
   I27 : BOOL ;
   I28 : BOOL ;
   I29 : BOOL ;
   I30 : BOOL ;
   I31 : BOOL ;
  END_STRUCT ;
END_VAR
BEGIN
NETWORK
TITLE =general

      SET   ;

// unit & equipment number ---------------------------------------------------
      L     DB1690.DBW    0;
      T     #UnitNo;

      L     DB1695.DBW   14;
      L     1000;
      *I    ;
      L     #UnitNo;
      +I    ;
      T     #EquipmentID;

// CIP ----------------------------------------------------------------------
      L     DB1695.DBW   18;
      L     0;
      <I    ;
      =     #CIP;

// Communicating Units-------------------------------------------------------
      L     DB1695.DBD   10;
      L     DB1695.DBD  106;
      ==D   ;
      =     #ComCIP;

// emergency OK -------------------------------------------------------------
      A     DB1695.DBX   75.0; //General Emergency Stop OK
      =     #EStopOK;

NETWORK
TITLE =read other unit's data

      SET   ;

// ... General Unit ----------/

      CALL FC   563 (
           ActReq                   := M    101.0,
           PLCNo                    := DB1695.DBW   14,
           SourceUnitNo             := 99,
           IsTUnit                  := FALSE,
           DstComDRec               := DB1695.GEN,
           RET_VAL                  := #wRetVal);


// ... CIP Unit ------------- /
      L     DB1691.DBD   46; // Select
      L     L#0; // Off
      ==D   ;
      JC    ELS1;
      TAK   ;
      L     DB1915.DBD   10; // CIP 1
      ==D   ;
      JC    M101;
      TAK   ;
      L     DB1925.DBD   10; // CIP 2
      ==D   ;
      JC    M102;
      TAK   ;
      L     DB1935.DBD   10; // CIP 3
      ==D   ;
      JC    M103;
      JU    ELS1;
M101: NOP   0; // Do 1
      CALL FC   563 (
           ActReq                   := M    101.0,
           PLCNo                    := 3,
           SourceUnitNo             := 91,
           IsTUnit                  := FALSE,
           DstComDRec               := DB1695.CIP,
           RET_VAL                  := #wRetVal);

      JU    FIN1;
M102: NOP   0; // Do 2
      CALL FC   563 (
           ActReq                   := M    101.0,
           PLCNo                    := 3,
           SourceUnitNo             := 92,
           IsTUnit                  := FALSE,
           DstComDRec               := DB1695.CIP,
           RET_VAL                  := #wRetVal);

      JU    FIN1;
M103: NOP   0; // Do 3
      CALL FC   563 (
           ActReq                   := M    101.0,
           PLCNo                    := 3,
           SourceUnitNo             := 93,
           IsTUnit                  := FALSE,
           DstComDRec               := DB1695.CIP,
           RET_VAL                  := #wRetVal);

      JU    FIN1;
ELS1: L     0;
      T     #iTmp;
      CALL SFC   21 (
           BVAL                     := #iTmp,
           RET_VAL                  := #iRetVal,
           BLK                      := DB1695.CIP);

FIN1: NOP   0;

NETWORK
TITLE =remote start
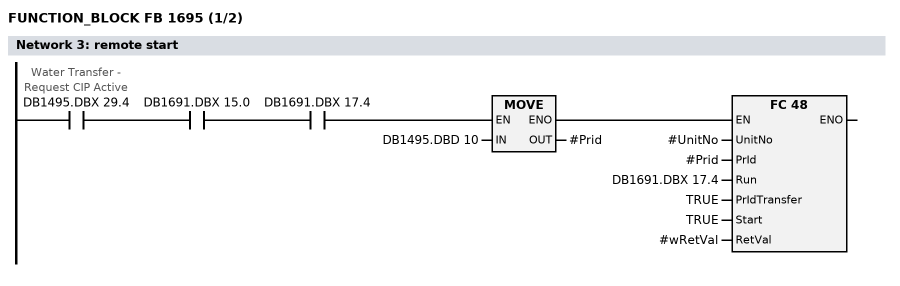

      SET   ;
      A     DB1495.DBX   29.4; // Water Transfer - Request CIP Active
      A     DB1691.DBX   15.0;
      A     DB1691.DBX   17.4;

      JCN   Strt;
      L     DB1495.DBD   10;
      T     #Prid;

      CALL FC    48 (
           UnitNo                   := #UnitNo,
           PrId                     := #Prid,
           Run                      := DB1691.DBX   17.4,
           PrIdTransfer             := TRUE,
           Start                    := TRUE,
           RetVal                   := #wRetVal);
Strt: NOP   0;
NETWORK
TITLE =external releases
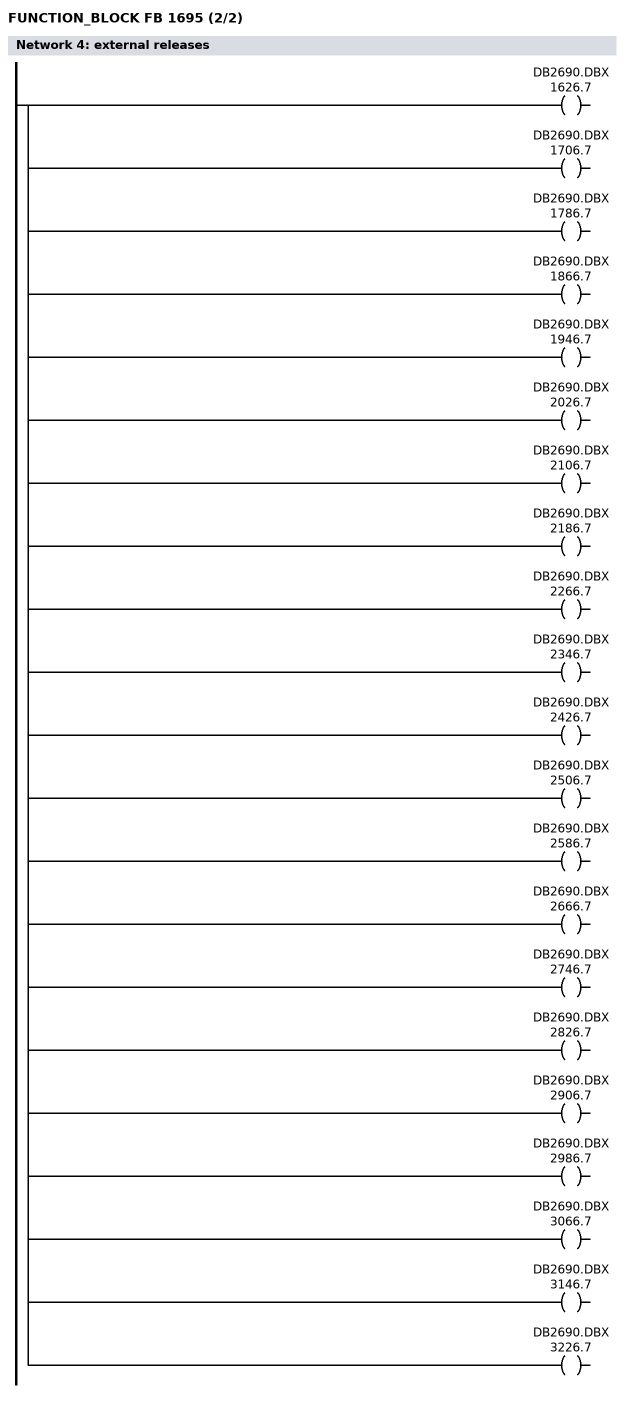

      SET   ;
      =     DB2690.DBX 1626.7;
      =     DB2690.DBX 1706.7;
      =     DB2690.DBX 1786.7;
      =     DB2690.DBX 1866.7;
      =     DB2690.DBX 1946.7;
      =     DB2690.DBX 2026.7;
      =     DB2690.DBX 2106.7;
      =     DB2690.DBX 2186.7;
      =     DB2690.DBX 2266.7;
      =     DB2690.DBX 2346.7;
      =     DB2690.DBX 2426.7;
      =     DB2690.DBX 2506.7;
      =     DB2690.DBX 2586.7;
      =     DB2690.DBX 2666.7;
      =     DB2690.DBX 2746.7;
      =     DB2690.DBX 2826.7;
      =     DB2690.DBX 2906.7;
      =     DB2690.DBX 2986.7;
      =     DB2690.DBX 3066.7;
      =     DB2690.DBX 3146.7;
      =     DB2690.DBX 3226.7;
NETWORK
TITLE =write own unit data

      SET   ;

//-- CIP Communication ---------------------------------------
      AN    DB1691.DBX   15.0;
      AN    DB1691.DBX 1233.6; // CIP Active (Slave)
      A     #ComCIP;
      JCN   NCIP;
//Conductivity CIP Return
      L     DB1695.DBD  150;
      T     DB1691.DBD  626;

//Temperature CIP Return
      L     DB1695.DBD  146;
      T     DB1691.DBD  594;

//CIP Prerun Pump SP

      CALL FC    45 (
           SFM                      := DB1691.DBD  686,
           Indexes                  := #SFM36);


      L     0.000000e+000;
      A     #SFM36.I01;
      =     DB1695.DBX  171.7;
      JCN   pfc;
      L     DB1691.DBD  654;
pfc:  NOP   0;
      A     #SFM36.I02;
      =     DB1695.DBX  172.0;
      JCN   ppc;
      L     DB1691.DBD  670;
ppc:  NOP   0;
      A     #SFM36.I03;
      =     DB1695.DBX  171.6;
      JCN   pxc;
      L     DB1691.DBD  574;
pxc:  NOP   0;
      T     DB1695.DBD  182;

//CIP Return
      L     DB1691.DBD  558;
      T     DB1695.DBD  186;
      L     DB1695.DBD  138;
      T     DB1691.DBD  562;

//CIP Prerun
      L     DB1691.DBD  542;
      T     DB1695.DBD  190;
      L     DB1695.DBD  142;
      T     DB1691.DBD  546;

// Write Own Data to CIP
      L     DB1695.DBD   10;
      T     DB1695.DBD  154;

      L     DB1695.DBW   14;
      T     DB1695.DBW  158;

      L     DB1695.DBW   16;
      T     DB1695.DBW  160;

      L     DB1695.DBW   18;
      T     DB1695.DBW  162;

      L     DB1695.DBW   20;
      T     DB1695.DBW  164;

      L     DB1695.DBW   22;
      T     DB1695.DBW  166;

      A     DB1695.DBX   24.0;
      =     DB1695.DBX  168.0;

      A     DB1695.DBX   24.1;
      =     DB1695.DBX  168.1;

      A     DB1695.DBX   24.2;
      =     DB1695.DBX  168.2;

      A     DB1695.DBX   24.3;
      =     DB1695.DBX  168.3;

      A     DB1695.DBX   24.4;
      =     DB1695.DBX  168.4;

      A     DB1695.DBX   24.5;
      =     DB1695.DBX  168.5;

      A     DB1695.DBX   24.6;
      =     DB1695.DBX  168.6;

      A     DB1695.DBX   24.7;
      =     DB1695.DBX  168.7;

// Copy Data to CIP
      CALL SFC   20 (
           SRCBLK                   := DB1695.ToCIP,
           RET_VAL                  := #iRetVal,
           DSTBLK                   := DB1695.ToCIP);

NCIP: NOP   0;

//Empty Signal
//A     "U069SpID".SpI.Sig //!!!! Insert correct Empty Signal !!!
      CLR   ;
      =     DB1695.DBX   26.5;

//Full Signal
//A     "U069SpID".SpI.Sig //!!!! Insert correct Full Signal !!!
      CLR   ;
      =     DB1695.DBX   26.2;

//CIP Program Selected
      A     #CIP;
      =     DB1695.DBX   27.1;

// Emergency Stop
      A     #EStopOK; //If needed add or replace with own SpI
      =     DB1695.DBX   27.0; //Emergency Stop OK


NETWORK
TITLE = read from other unit data



END_FUNCTION_BLOCK

FUNCTION_BLOCK FB 1699
TITLE =U069: Packaging Plant 9
AUTHOR : Woermann
FAMILY : BOTEC_F1
NAME : Sim
VERSION : 0.1


VAR_TEMP
  CIP : BOOL ;	//CIP active
  xTmp : BOOL ;	//Temporary BOOL (free for general use)
  iTmp : INT ;	//Temporary INT (free for general use)
  rTmp : REAL ;	//Temporary REAL (free for general use)
  UnitNo : INT ;	//Unit Number
END_VAR
BEGIN
NETWORK
TITLE =General

      SET   ;
// get unit number ----------------------------------------------------------
      L     DB1690.DBW    0;
      T     #UnitNo;

// CIP ----------------------------------------------------------------------
      L     DB1691.DBD   54;
      L     0;
      <D    ;
      =     #CIP;

NETWORK
TITLE =Actuator

      A     DB1691.DBX   17.3;
      =     DB2690.DBX 1625.3;
      =     DB2690.DBX 1705.3;
      =     DB2690.DBX 1785.3;
      =     DB2690.DBX 1865.3;
      =     DB2690.DBX 1945.3;
      =     DB2690.DBX 2025.3;
      =     DB2690.DBX 2105.3;
      =     DB2690.DBX 2185.3;
      =     DB2690.DBX 2265.3;
      =     DB2690.DBX 2345.3;
      =     DB2690.DBX 2425.3;
      =     DB2690.DBX 2505.3;
      =     DB2690.DBX 2585.3;
      =     DB2690.DBX 2665.3;
      =     DB2690.DBX 2745.3;
      =     DB2690.DBX 2825.3;
      =     DB2690.DBX 2905.3;
      =     DB2690.DBX 2985.3;
      =     DB2690.DBX 3065.3;
      =     DB2690.DBX 3145.3;
      =     DB2690.DBX 3225.3;

NETWORK
TITLE =Special Input

      A     DB1691.DBX   17.3;
      =     DB2691.DBX   81.3;
      =     DB2691.DBX  141.3;
      =     DB2691.DBX  441.3;
      =     DB2691.DBX  501.3;
      =     DB2691.DBX  561.3;
      =     DB2691.DBX  621.3;
      =     DB2691.DBX  681.3;
      =     DB2691.DBX  741.3;
      =     DB2691.DBX  801.3;
      =     DB2691.DBX  861.3;
      =     DB2691.DBX  921.3;
      =     DB2691.DBX  981.3;
      =     DB2691.DBX 1041.3;
      =     DB2691.DBX 1101.3;
      =     DB2691.DBX 1161.3;
      =     DB2691.DBX 1221.3;
      =     DB2691.DBX 1281.3;
      =     DB2691.DBX 1341.3;
      =     DB2691.DBX 1401.3;
      =     DB2691.DBX 1461.3;
      =     DB2691.DBX 1521.3;

NETWORK
TITLE =Counter

      A     DB1691.DBX   17.3;
      A     M    101.0;


      CLR   ;
NETWORK
TITLE =Analog Input

      A     DB1691.DBX   17.3;
      =     DB2693.DBX  141.3;

NETWORK
TITLE =Universal Value

      A     DB1691.DBX   17.3;
//      =     "U069UnVD".unv001.Sim;
//      =     "U069UnVD".unv002.Sim;
//      =     "U069UnVD".unv003.Sim;
//      =     "U069UnVD".unv004.Sim;

NETWORK
TITLE =PID

      A     DB1691.DBX   17.3;

NETWORK
TITLE =Message

      A     DB1691.DBX   17.3;
//      =     "U069MsgD".msg001.Sim;
//      =     "U069MsgD".msg002.Sim;
//      =     "U069MsgD".msg003.Sim;

NETWORK
TITLE =VLT

      A     DB1691.DBX   17.3;

END_FUNCTION_BLOCK

FUNCTION_BLOCK FB 1705
TITLE =U070: Packaging Plant 10
FAMILY : BOTEC_F1
NAME : Comm
VERSION : 0.1


VAR_TEMP
  iRetVal : INT ;	//return value as integer
  wRetVal : WORD ;	//return value as word
  Run : BOOL ;	//Unit in "RUN" mode
  EStopOK : BOOL ;	//Emergency Stop OK
  CIP : BOOL ;	//CIP Program Selected
  ComCIP : BOOL ;	//Communication with CIP Active
  xTmp : BOOL ;	//Temporary BOOL (free for general use)
  iTmp : INT ;	//Temporary INT (free for general use)
  rTmp : REAL ;	//Temporary REAL (free for general use)
  dTmp : DINT ;	//Temporary DINT (free for general use)
  UnitNo : INT ;	//Unit Number
  EquipmentID : INT ;	//Equipment ID
  Prid : DINT ;	//Process ID
  SFM36 : STRUCT 	// CIP Pump Mode
   I00 : BOOL ;	// Off
   I01 : BOOL ;	// Flow
   I02 : BOOL ;	// Pressure
   I03 : BOOL ;	// Fix Speed
   I04 : BOOL ;
   I05 : BOOL ;
   I06 : BOOL ;
   I07 : BOOL ;
   I08 : BOOL ;
   I09 : BOOL ;
   I10 : BOOL ;
   I11 : BOOL ;
   I12 : BOOL ;
   I13 : BOOL ;
   I14 : BOOL ;
   I15 : BOOL ;
   I16 : BOOL ;
   I17 : BOOL ;
   I18 : BOOL ;
   I19 : BOOL ;
   I20 : BOOL ;
   I21 : BOOL ;
   I22 : BOOL ;
   I23 : BOOL ;
   I24 : BOOL ;
   I25 : BOOL ;
   I26 : BOOL ;
   I27 : BOOL ;
   I28 : BOOL ;
   I29 : BOOL ;
   I30 : BOOL ;
   I31 : BOOL ;
  END_STRUCT ;
END_VAR
BEGIN
NETWORK
TITLE =general

      SET   ;

// unit & equipment number ---------------------------------------------------
      L     DB1700.DBW    0;
      T     #UnitNo;

      L     DB1705.DBW   14;
      L     1000;
      *I    ;
      L     #UnitNo;
      +I    ;
      T     #EquipmentID;

// CIP ----------------------------------------------------------------------
      L     DB1705.DBW   18;
      L     0;
      <I    ;
      =     #CIP;

// Communicating Units-------------------------------------------------------
      L     DB1705.DBD   10;
      L     DB1705.DBD  106;
      ==D   ;
      =     #ComCIP;

// emergency OK -------------------------------------------------------------
      A     DB1705.DBX   75.0; //General Emergency Stop OK
      =     #EStopOK;

NETWORK
TITLE =read other unit's data

      SET   ;

// ... General Unit ----------/

      CALL FC   563 (
           ActReq                   := M    101.0,
           PLCNo                    := DB1705.DBW   14,
           SourceUnitNo             := 99,
           IsTUnit                  := FALSE,
           DstComDRec               := DB1705.GEN,
           RET_VAL                  := #wRetVal);


// ... CIP Unit ------------- /
      L     DB1701.DBD   46; // Select
      L     L#0; // Off
      ==D   ;
      JC    ELS1;
      TAK   ;
      L     DB1915.DBD   10; // CIP 1
      ==D   ;
      JC    M101;
      TAK   ;
      L     DB1925.DBD   10; // CIP 2
      ==D   ;
      JC    M102;
      TAK   ;
      L     DB1935.DBD   10; // CIP 3
      ==D   ;
      JC    M103;
      JU    ELS1;
M101: NOP   0; // Do 1
      CALL FC   563 (
           ActReq                   := M    101.0,
           PLCNo                    := 3,
           SourceUnitNo             := 91,
           IsTUnit                  := FALSE,
           DstComDRec               := DB1705.CIP,
           RET_VAL                  := #wRetVal);

      JU    FIN1;
M102: NOP   0; // Do 2
      CALL FC   563 (
           ActReq                   := M    101.0,
           PLCNo                    := 3,
           SourceUnitNo             := 92,
           IsTUnit                  := FALSE,
           DstComDRec               := DB1705.CIP,
           RET_VAL                  := #wRetVal);

      JU    FIN1;
M103: NOP   0; // Do 3
      CALL FC   563 (
           ActReq                   := M    101.0,
           PLCNo                    := 3,
           SourceUnitNo             := 93,
           IsTUnit                  := FALSE,
           DstComDRec               := DB1705.CIP,
           RET_VAL                  := #wRetVal);

      JU    FIN1;
ELS1: L     0;
      T     #iTmp;
      CALL SFC   21 (
           BVAL                     := #iTmp,
           RET_VAL                  := #iRetVal,
           BLK                      := DB1705.CIP);

FIN1: NOP   0;

NETWORK
TITLE =remote start
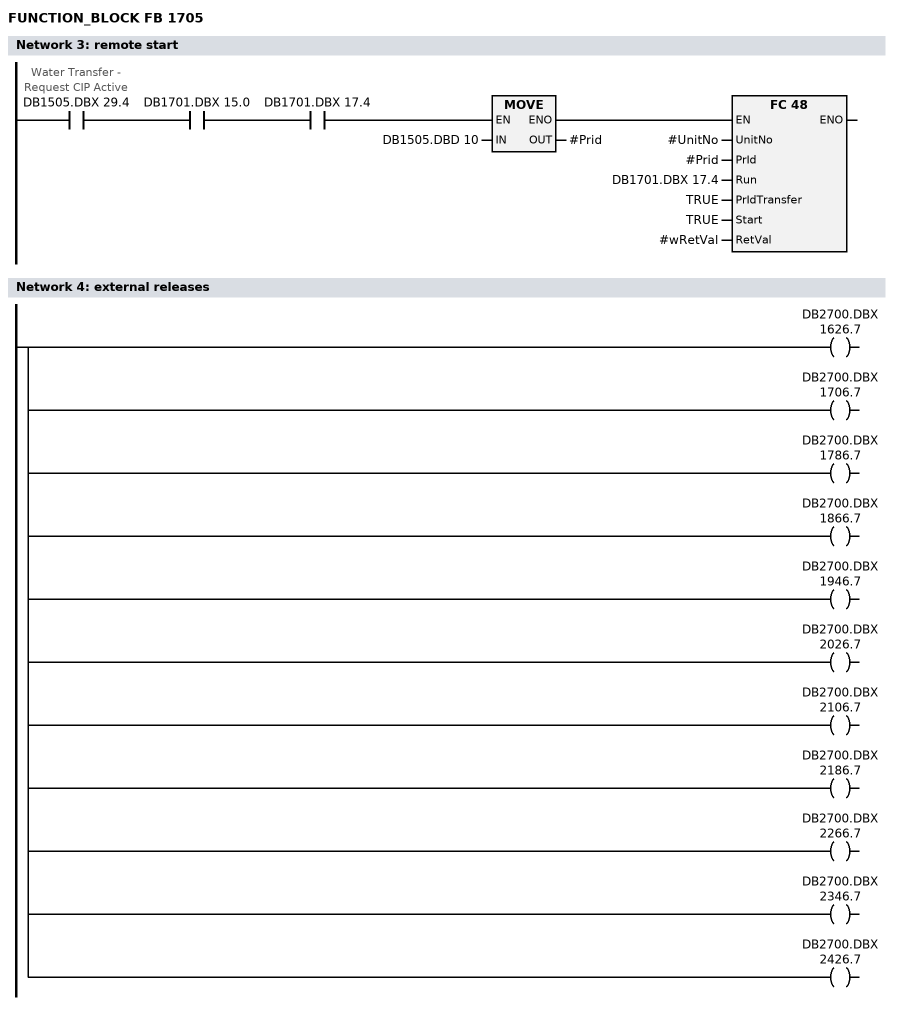

      SET   ;
      A     DB1505.DBX   29.4; // Water Transfer - Request CIP Active
      A     DB1701.DBX   15.0;
      A     DB1701.DBX   17.4;

      JCN   Strt;
      L     DB1505.DBD   10;
      T     #Prid;

      CALL FC    48 (
           UnitNo                   := #UnitNo,
           PrId                     := #Prid,
           Run                      := DB1701.DBX   17.4,
           PrIdTransfer             := TRUE,
           Start                    := TRUE,
           RetVal                   := #wRetVal);
Strt: NOP   0;
NETWORK
TITLE =external releases

      SET   ;
      =     DB2700.DBX 1626.7;
      =     DB2700.DBX 1706.7;
      =     DB2700.DBX 1786.7;
      =     DB2700.DBX 1866.7;
      =     DB2700.DBX 1946.7;
      =     DB2700.DBX 2026.7;
      =     DB2700.DBX 2106.7;
      =     DB2700.DBX 2186.7;
      =     DB2700.DBX 2266.7;
      =     DB2700.DBX 2346.7;
      =     DB2700.DBX 2426.7;
NETWORK
TITLE =write own unit data

      SET   ;

//-- CIP Communication ---------------------------------------
      AN    DB1701.DBX   15.0;
//      AN "U070SeqD".Seq.PO.B30 // CIP Active (Slave)
      A     #ComCIP;
      JCN   NCIP;
//Conductivity CIP Return
      L     DB1705.DBD  150;
      T     DB1701.DBD  626;

//Temperature CIP Return
      L     DB1705.DBD  146;
      T     DB1701.DBD  594;

//CIP Prerun Pump SP

      CALL FC    45 (
           SFM                      := DB1701.DBD  686,
           Indexes                  := #SFM36);


      L     0.000000e+000;
      A     #SFM36.I01;
      =     DB1705.DBX  171.7;
      JCN   pfc;
      L     DB1701.DBD  654;
pfc:  NOP   0;
      A     #SFM36.I02;
      =     DB1705.DBX  172.0;
      JCN   ppc;
      L     DB1701.DBD  670;
ppc:  NOP   0;
      A     #SFM36.I03;
      =     DB1705.DBX  171.6;
      JCN   pxc;
      L     DB1701.DBD  574;
pxc:  NOP   0;
      T     DB1705.DBD  182;

//CIP Return
      L     DB1701.DBD  558;
      T     DB1705.DBD  186;
      L     DB1705.DBD  138;
      T     DB1701.DBD  562;

//CIP Prerun
      L     DB1701.DBD  542;
      T     DB1705.DBD  190;
      L     DB1705.DBD  142;
      T     DB1701.DBD  546;

// Write Own Data to CIP
      L     DB1705.DBD   10;
      T     DB1705.DBD  154;

      L     DB1705.DBW   14;
      T     DB1705.DBW  158;

      L     DB1705.DBW   16;
      T     DB1705.DBW  160;

      L     DB1705.DBW   18;
      T     DB1705.DBW  162;

      L     DB1705.DBW   20;
      T     DB1705.DBW  164;

      L     DB1705.DBW   22;
      T     DB1705.DBW  166;

      A     DB1705.DBX   24.0;
      =     DB1705.DBX  168.0;

      A     DB1705.DBX   24.1;
      =     DB1705.DBX  168.1;

      A     DB1705.DBX   24.2;
      =     DB1705.DBX  168.2;

      A     DB1705.DBX   24.3;
      =     DB1705.DBX  168.3;

      A     DB1705.DBX   24.4;
      =     DB1705.DBX  168.4;

      A     DB1705.DBX   24.5;
      =     DB1705.DBX  168.5;

      A     DB1705.DBX   24.6;
      =     DB1705.DBX  168.6;

      A     DB1705.DBX   24.7;
      =     DB1705.DBX  168.7;

// Copy Data to CIP
      CALL SFC   20 (
           SRCBLK                   := DB1705.ToCIP,
           RET_VAL                  := #iRetVal,
           DSTBLK                   := DB1705.ToCIP);

NCIP: NOP   0;

//Empty Signal
//A     "U070SpID".SpI.Sig //!!!! Insert correct Empty Signal !!!
      CLR   ;
      =     DB1705.DBX   26.5;

//Full Signal
//A     "U070SpID".SpI.Sig //!!!! Insert correct Full Signal !!!
      CLR   ;
      =     DB1705.DBX   26.2;

//CIP Program Selected
      A     #CIP;
      =     DB1705.DBX   27.1;

// Emergency Stop
      A     #EStopOK; //If needed add or replace with own SpI
      =     DB1705.DBX   27.0; //Emergency Stop OK


NETWORK
TITLE = read from other unit data



END_FUNCTION_BLOCK

FUNCTION_BLOCK FB 1709
TITLE =U070: Packaging Plant 10
AUTHOR : Woermann
FAMILY : BOTEC_F1
NAME : Sim
VERSION : 0.1


VAR_TEMP
  CIP : BOOL ;	//CIP active
  xTmp : BOOL ;	//Temporary BOOL (free for general use)
  iTmp : INT ;	//Temporary INT (free for general use)
  rTmp : REAL ;	//Temporary REAL (free for general use)
  UnitNo : INT ;	//Unit Number
END_VAR
BEGIN
NETWORK
TITLE =General

      SET   ;
// get unit number ----------------------------------------------------------
      L     DB1700.DBW    0;
      T     #UnitNo;

// CIP ----------------------------------------------------------------------
      L     DB1701.DBD   54;
      L     0;
      <D    ;
      =     #CIP;

NETWORK
TITLE =Actuator

      A     DB1701.DBX   17.3;
      =     DB2700.DBX 1625.3;
      =     DB2700.DBX 1705.3;
      =     DB2700.DBX 1785.3;
      =     DB2700.DBX 1865.3;
      =     DB2700.DBX 1945.3;
      =     DB2700.DBX 2025.3;
      =     DB2700.DBX 2105.3;
      =     DB2700.DBX 2185.3;
      =     DB2700.DBX 2265.3;
      =     DB2700.DBX 2345.3;
      =     DB2700.DBX 2425.3;

NETWORK
TITLE =Special Input

      A     DB1701.DBX   17.3;
      =     DB2701.DBX   81.3;
      =     DB2701.DBX  141.3;
      =     DB2701.DBX  201.3;
      =     DB2701.DBX  261.3;
      =     DB2701.DBX  321.3;
      =     DB2701.DBX  381.3;
      =     DB2701.DBX  441.3;
      =     DB2701.DBX  501.3;
      =     DB2701.DBX  561.3;
      =     DB2701.DBX  621.3;

NETWORK
TITLE =Counter

      A     DB1701.DBX   17.3;
      A     M    101.0;


      CLR   ;
NETWORK
TITLE =Analog Input

      A     DB1701.DBX   17.3;

NETWORK
TITLE =Universal Value

      A     DB1701.DBX   17.3;
//      =     "U070UnVD".unv001.Sim;
//      =     "U070UnVD".unv002.Sim;
//      =     "U070UnVD".unv003.Sim;
//      =     "U070UnVD".unv004.Sim;

NETWORK
TITLE =PID

      A     DB1701.DBX   17.3;

NETWORK
TITLE =Message

      A     DB1701.DBX   17.3;
//      =     "U070MsgD".msg001.Sim;
//      =     "U070MsgD".msg002.Sim;
//      =     "U070MsgD".msg003.Sim;

NETWORK
TITLE =VLT

      A     DB1701.DBX   17.3;

END_FUNCTION_BLOCK

FUNCTION_BLOCK FB 1715
TITLE =U071: Packaging Plant 11
FAMILY : BOTEC_F1
NAME : Comm
VERSION : 0.1


VAR_TEMP
  iRetVal : INT ;	//return value as integer
  wRetVal : WORD ;	//return value as word
  Run : BOOL ;	//Unit in "RUN" mode
  EStopOK : BOOL ;	//Emergency Stop OK
  CIP : BOOL ;	//CIP Program Selected
  ComCIP : BOOL ;	//Communication with CIP Active
  xTmp : BOOL ;	//Temporary BOOL (free for general use)
  iTmp : INT ;	//Temporary INT (free for general use)
  rTmp : REAL ;	//Temporary REAL (free for general use)
  dTmp : DINT ;	//Temporary DINT (free for general use)
  UnitNo : INT ;	//Unit Number
  EquipmentID : INT ;	//Equipment ID
  Prid : DINT ;	//Process ID
  SFM36 : STRUCT 	// CIP Pump Mode
   I00 : BOOL ;	// Off
   I01 : BOOL ;	// Flow
   I02 : BOOL ;	// Pressure
   I03 : BOOL ;	// Fix Speed
   I04 : BOOL ;
   I05 : BOOL ;
   I06 : BOOL ;
   I07 : BOOL ;
   I08 : BOOL ;
   I09 : BOOL ;
   I10 : BOOL ;
   I11 : BOOL ;
   I12 : BOOL ;
   I13 : BOOL ;
   I14 : BOOL ;
   I15 : BOOL ;
   I16 : BOOL ;
   I17 : BOOL ;
   I18 : BOOL ;
   I19 : BOOL ;
   I20 : BOOL ;
   I21 : BOOL ;
   I22 : BOOL ;
   I23 : BOOL ;
   I24 : BOOL ;
   I25 : BOOL ;
   I26 : BOOL ;
   I27 : BOOL ;
   I28 : BOOL ;
   I29 : BOOL ;
   I30 : BOOL ;
   I31 : BOOL ;
  END_STRUCT ;
END_VAR
BEGIN
NETWORK
TITLE =general

      SET   ;

// unit & equipment number ---------------------------------------------------
      L     DB1710.DBW    0;
      T     #UnitNo;

      L     DB1715.DBW   14;
      L     1000;
      *I    ;
      L     #UnitNo;
      +I    ;
      T     #EquipmentID;

// CIP ----------------------------------------------------------------------
      L     DB1715.DBW   18;
      L     0;
      <I    ;
      =     #CIP;

